C01810=1065.952,131.277,423.591,172.677,28.451,155.205
C01811=1065.946,131.028,423.611,172.676,28.448,155.204
C01812=1065.940,130.779,423.631,172.674,28.445,155.204
C01813=1065.934,130.529,423.652,172.673,28.443,155.203
C01814=1065.928,130.280,423.672,172.671,28.440,155.203
C01815=1065.922,130.032,423.692,172.669,28.438,155.203
C01816=1065.917,129.783,423.712,172.667,28.435,155.202
C01817=1065.911,129.533,423.733,172.665,28.432,155.202
C01818=1065.905,129.284,423.753,172.664,28.429,155.201
C01819=1065.899,129.035,423.772,172.662,28.426,155.201
C01820=1065.894,128.786,423.792,172.660,28.424,155.201
C01821=1065.887,128.536,423.813,172.659,28.421,155.200
C01822=1065.881,128.287,423.833,172.657,28.418,155.200
C01823=1065.876,128.038,423.853,172.656,28.416,155.200
C01824=1065.870,127.789,423.873,172.654,28.413,155.199
C01825=1065.863,127.540,423.894,172.652,28.410,155.199
C01826=1065.857,127.291,423.914,172.651,28.408,155.198
C01827=1065.851,127.007,423.936,172.648,28.404,155.198
C01828=1065.845,126.724,423.959,172.647,28.401,155.197
C01829=1065.837,126.440,423.982,172.645,28.398,155.197
C01830=1065.831,126.157,424.005,172.643,28.395,155.197
C01831=1065.826,125.907,424.025,172.641,28.392,155.196
C01832=1065.820,125.658,424.045,172.640,28.390,155.196
C01833=1065.814,125.409,424.065,172.638,28.387,155.195
C01834=1065.807,125.160,424.085,172.636,28.384,155.195
C01835=1065.802,124.911,424.106,172.635,28.381,155.195
C01836=1065.796,124.662,424.126,172.633,28.379,155.194
C01837=1065.790,124.412,424.145,172.632,28.376,155.194
C01838=1065.784,124.164,424.165,172.630,28.373,155.193
C01839=1065.779,123.914,424.186,172.628,28.370,155.193
C01840=1065.772,123.665,424.206,172.627,28.368,155.193
C01841=1065.767,123.416,424.225,172.625,28.365,155.192
C01842=1065.761,123.167,424.245,172.624,28.363,155.192
C01843=1065.755,122.918,424.265,172.622,28.360,155.191
C01844=1065.749,122.669,424.286,172.620,28.357,155.191
C01845=1065.744,122.419,424.305,172.619,28.354,155.191
C01846=1065.738,122.171,424.325,172.617,28.352,155.190
C01847=1065.732,121.922,424.345,172.616,28.349,155.190
C01848=1065.727,121.672,424.365,172.614,28.346,155.189
C01849=1065.721,121.423,424.385,172.612,28.343,155.189
C01850=1065.714,121.174,424.405,172.610,28.340,155.189
C01851=1065.708,120.924,424.424,172.608,28.337,155.188
C01852=1065.702,120.675,424.444,172.607,28.335,155.188
C01853=1065.697,120.426,424.465,172.605,28.332,155.187
C01854=1065.692,120.177,424.484,172.604,28.329,155.187
C01855=1065.686,119.928,424.504,172.602,28.326,155.187
C01856=1065.680,119.679,424.524,172.601,28.324,155.186
C01857=1065.674,119.430,424.543,172.599,28.321,155.186
C01858=1065.669,119.181,424.564,172.597,28.318,155.185
C01859=1065.663,118.931,424.583,172.596,28.315,155.185
C01860=1065.657,118.682,424.603,172.594,28.313,155.185
C01861=1065.651,118.434,424.623,172.593,28.310,155.184
C01862=1065.645,118.184,424.642,172.591,28.307,155.184
C01863=1065.639,117.935,424.662,172.589,28.304,155.183
C01864=1065.634,117.686,424.682,172.588,28.302,155.183
C01865=1065.628,117.437,424.702,172.586,28.299,155.183
C01866=1065.623,117.187,424.721,172.585,28.296,155.182
C01867=1065.617,116.939,424.741,172.583,28.293,155.182
C01868=1065.611,116.689,424.760,172.582,28.291,155.181
C01869=1065.605,116.440,424.780,172.580,28.288,155.181
C01870=1065.600,116.191,424.800,172.578,28.285,155.181
C01871=1065.594,115.942,424.820,172.577,28.282,155.180
C01872=1065.588,115.692,424.839,172.575,28.280,155.180
C01873=1065.582,115.444,424.859,172.574,28.277,155.179
C01874=1065.577,115.194,424.878,172.572,28.274,155.179
C01875=1065.571,114.945,424.898,172.571,28.271,155.178
C01876=1065.565,114.696,424.918,172.569,28.268,155.178
C01877=1065.560,114.447,424.938,172.568,28.265,155.178
C01878=1065.554,114.197,424.957,172.566,28.262,155.177
C01879=1065.548,113.948,424.977,172.564,28.260,155.177
C01880=1065.542,113.699,424.997,172.563,28.257,155.176
C01881=1065.537,113.450,425.016,172.561,28.255,155.176
C01882=1065.530,113.201,425.035,172.560,28.252,155.176
C01883=1065.524,112.952,425.054,172.558,28.249,155.175
C01884=1065.519,112.702,425.074,172.556,28.246,155.175
C01885=1065.513,112.453,425.094,172.555,28.244,155.174
C01886=1065.507,112.204,425.113,172.553,28.241,155.174
C01887=1065.501,111.955,425.132,172.552,28.238,155.174
C01888=1065.495,111.706,425.152,172.550,28.235,155.173
C01889=1065.489,111.456,425.171,172.549,28.232,155.173
C01890=1065.484,111.207,425.191,172.547,28.230,155.172
C01891=1065.477,110.923,425.213,172.545,28.227,155.172
C01892=1065.470,110.640,425.235,172.543,28.223,155.172
C01893=1065.463,110.356,425.257,172.541,28.221,155.171
C01894=1065.457,110.072,425.279,172.540,28.217,155.171
C01895=1065.450,109.823,425.298,172.538,28.215,155.170
C01896=1065.445,109.574,425.317,172.537,28.212,155.170
C01897=1065.439,109.325,425.336,172.535,28.210,155.170
C01898=1065.433,109.075,425.356,172.534,28.207,155.169
C01899=1065.427,108.826,425.376,172.532,28.204,155.169
C01900=1065.421,108.577,425.394,172.530,28.201,155.168
C01901=1065.415,108.328,425.414,172.529,28.198,155.168
C01902=1065.410,108.078,425.433,172.527,28.196,155.168
C01903=1065.404,107.830,425.452,172.526,28.193,155.167
C01904=1065.398,107.581,425.471,172.524,28.190,155.167
C01905=1065.392,107.332,425.490,172.523,28.187,155.166
C01906=1065.386,107.082,425.510,172.521,28.185,155.166
C01907=1065.381,106.833,425.529,172.519,28.182,155.166
C01908=1065.374,106.584,425.547,172.518,28.180,155.165
C01909=1065.369,106.334,425.567,172.516,28.177,155.165
C01910=1065.363,106.085,425.586,172.515,28.174,155.164
C01911=1065.357,105.836,425.606,172.513,28.171,155.164
C01912=1065.350,105.587,425.625,172.512,28.169,155.164
C01913=1065.345,105.338,425.643,172.510,28.166,155.163
C01914=1065.340,105.089,425.663,172.508,28.163,155.163
C01915=1065.334,104.839,425.682,172.507,28.160,155.162
C01916=1065.328,104.590,425.701,172.505,28.157,155.162
C01917=1065.322,104.341,425.720,172.504,28.155,155.162
C01918=1065.316,104.091,425.739,172.502,28.152,155.161
C01919=1065.310,103.842,425.758,172.501,28.149,155.161
C01920=1065.305,103.593,425.777,172.499,28.146,155.160
C01921=1065.299,103.344,425.796,172.498,28.144,155.160
C01922=1065.293,103.095,425.815,172.497,28.141,155.160
C01923=1065.287,102.845,425.834,172.495,28.138,155.159
C01924=1065.281,102.596,425.853,172.494,28.136,155.159
C01925=1065.275,102.347,425.872,172.492,28.133,155.158
C01926=1065.270,102.098,425.890,172.491,28.130,155.158
C01927=1065.264,101.849,425.910,172.489,28.127,155.158
C01928=1065.258,101.599,425.929,172.488,28.124,155.157
C01929=1065.253,101.350,425.948,172.486,28.122,155.157
C01930=1065.246,101.101,425.967,172.484,28.119,155.156
C01931=1065.241,100.852,425.986,172.483,28.116,155.156
C01932=1065.235,100.603,426.004,172.481,28.114,155.156
C01933=1065.229,100.353,426.024,172.480,28.111,155.155
C01934=1065.223,100.104,426.042,172.478,28.108,155.155
C01935=1065.217,99.855,426.061,172.477,28.106,155.154
C01936=1065.210,99.606,426.080,172.475,28.103,155.154
C01937=1065.205,99.356,426.099,172.473,28.100,155.154
C01938=1065.199,99.108,426.118,172.472,28.097,155.153
C01939=1065.193,98.859,426.137,172.470,28.094,155.153
C01940=1065.187,98.609,426.155,172.469,28.092,155.153
C01941=1065.181,98.359,426.174,172.467,28.089,155.152
C01942=1065.175,98.110,426.193,172.466,28.087,155.152
C01943=1065.170,97.862,426.212,172.464,28.084,155.151
C01944=1065.163,97.612,426.230,172.462,28.081,155.151
C01945=1065.158,97.363,426.249,172.461,28.078,155.151
C01946=1065.151,97.114,426.268,172.460,28.076,155.150
C01947=1065.146,96.864,426.287,172.459,28.073,155.150
C01948=1065.140,96.615,426.305,172.457,28.070,155.149
C01949=1065.134,96.366,426.324,172.456,28.067,155.149
C01950=1065.128,96.117,426.343,172.454,28.065,155.149
C01951=1065.122,95.867,426.361,172.452,28.062,155.148
C01952=1065.117,95.618,426.380,172.451,28.060,155.148
C01953=1065.110,95.369,426.398,172.449,28.057,155.147
C01954=1065.105,95.120,426.418,172.448,28.054,155.147
C01955=1065.098,94.836,426.439,172.446,28.051,155.147
C01956=1065.091,94.553,426.459,172.445,28.048,155.146
C01957=1065.085,94.268,426.481,172.442,28.044,155.146
C01958=1065.078,93.985,426.503,172.441,28.042,155.145
C01959=1065.072,93.736,426.520,172.439,28.039,155.145
C01960=1065.067,93.486,426.539,172.438,28.036,155.144
C01961=1065.060,93.237,426.558,172.436,28.033,155.144
C01962=1065.055,92.988,426.576,172.435,28.030,155.144
C01963=1065.049,92.739,426.595,172.433,28.028,155.143
C01964=1065.043,92.490,426.613,172.431,28.025,155.143
C01965=1065.037,92.240,426.632,172.431,28.022,155.142
C01966=1065.031,91.991,426.650,172.429,28.020,155.142
C01967=1065.026,91.742,426.670,172.428,28.017,155.142
C01968=1065.020,91.492,426.687,172.426,28.014,155.141
C01969=1065.014,91.244,426.706,172.425,28.011,155.141
C01970=1065.008,90.994,426.725,172.423,28.009,155.141
C01971=1065.002,90.745,426.743,172.421,28.006,155.140
C01972=1064.996,90.496,426.761,172.420,28.003,155.140
C01973=1064.991,90.246,426.780,172.418,28.001,155.139
C01974=1064.984,89.997,426.798,172.417,27.998,155.139
C01975=1064.979,89.748,426.816,172.415,27.995,155.139
C01976=1064.972,89.499,426.835,172.414,27.992,155.138
C01977=1064.966,89.250,426.853,172.412,27.990,155.138
C01978=1064.961,89.000,426.872,172.410,27.987,155.137
C01979=1064.955,88.751,426.890,172.409,27.985,155.137
C01980=1064.949,88.501,426.908,172.408,27.982,155.137
C01981=1064.942,88.252,426.927,172.407,27.979,155.136
C01982=1064.937,88.003,426.944,172.405,27.976,155.136
C01983=1064.931,87.754,426.963,172.404,27.974,155.135
C01984=1064.925,87.504,426.981,172.402,27.971,155.135
C01985=1064.919,87.256,427.000,172.401,27.969,155.135
C01986=1064.913,87.006,427.018,172.399,27.966,155.134
C01987=1064.906,86.757,427.036,172.397,27.963,155.134
C01988=1064.901,86.508,427.054,172.396,27.960,155.134
C01989=1064.896,86.258,427.072,172.394,27.957,155.133
C01990=1064.889,86.009,427.091,172.393,27.955,155.133
C01991=1064.884,85.760,427.109,172.391,27.952,155.132
C01992=1064.877,85.510,427.127,172.390,27.949,155.132
C01993=1064.871,85.261,427.145,172.388,27.947,155.132
C01994=1064.865,85.012,427.163,172.387,27.944,155.131
C01995=1064.859,84.763,427.181,172.386,27.942,155.131
C01996=1064.854,84.513,427.200,172.384,27.939,155.130
C01997=1064.848,84.264,427.218,172.383,27.936,155.130
C01998=1064.842,84.014,427.236,172.381,27.933,155.130
C01999=1064.836,83.766,427.254,172.380,27.930,155.129
C02000=1064.830,83.516,427.272,172.378,27.928,155.129
C02001=1064.824,83.267,427.290,172.377,27.925,155.128
C02002=1064.818,83.018,427.309,172.375,27.922,155.128
C02003=1064.812,82.768,427.326,172.373,27.920,155.128
C02004=1064.807,82.519,427.345,172.372,27.917,155.127
C02005=1064.801,82.270,427.363,172.370,27.914,155.127
C02006=1064.795,82.021,427.381,172.370,27.912,155.127
C02007=1064.789,81.771,427.399,172.368,27.909,155.126
C02008=1064.783,81.522,427.416,172.367,27.906,155.126
C02009=1064.777,81.273,427.435,172.365,27.903,155.125
C02010=1064.771,81.024,427.453,172.364,27.900,155.125
C02011=1064.765,80.774,427.470,172.362,27.898,155.125
C02012=1064.760,80.526,427.489,172.361,27.895,155.124
C02013=1064.754,80.276,427.507,172.359,27.892,155.124
C02014=1064.748,80.026,427.525,172.357,27.889,155.123
C02015=1064.743,79.777,427.543,172.356,27.887,155.123
C02016=1064.736,79.528,427.561,172.354,27.884,155.123
C02017=1064.731,79.279,427.579,172.354,27.882,155.122
C02018=1064.724,79.029,427.597,172.352,27.879,155.122
C02019=1064.718,78.746,427.618,172.350,27.875,155.121
C02020=1064.711,78.462,427.637,172.348,27.873,155.121
C02021=1064.704,78.178,427.658,172.347,27.869,155.120
C02022=1064.698,77.894,427.678,172.345,27.866,155.120
C02023=1064.692,77.645,427.697,172.344,27.864,155.120
C02024=1064.686,77.396,427.714,172.342,27.861,155.119
C02025=1064.680,77.146,427.732,172.341,27.858,155.119
C02026=1064.674,76.898,427.749,172.339,27.855,155.118
C02027=1064.668,76.648,427.767,172.338,27.853,155.118
C02028=1064.662,76.399,427.784,172.336,27.850,155.118
C02029=1064.656,76.149,427.802,172.335,27.848,155.117
C02030=1064.650,75.901,427.821,172.334,27.845,155.117
C02031=1064.644,75.651,427.839,172.332,27.842,155.117
C02032=1064.639,75.402,427.856,172.331,27.839,155.116
C02033=1064.633,75.152,427.874,172.329,27.836,155.116
C02034=1064.626,74.903,427.891,172.328,27.834,155.115
C02035=1064.620,74.654,427.909,172.326,27.831,155.115
C02036=1064.615,74.405,427.927,172.325,27.829,155.115
C02037=1064.609,74.155,427.945,172.323,27.826,155.114
C02038=1064.603,73.906,427.962,172.321,27.823,155.114
C02039=1064.597,73.656,427.980,172.321,27.820,155.113
C02040=1064.591,73.407,427.998,172.319,27.818,155.113
C02041=1064.585,73.158,428.015,172.318,27.815,155.113
C02042=1064.579,72.909,428.033,172.316,27.813,155.112
C02043=1064.573,72.659,428.050,172.315,27.810,155.112
C02044=1064.567,72.410,428.068,172.313,27.807,155.112
C02045=1064.561,72.160,428.086,172.312,27.804,155.111
C02046=1064.556,71.911,428.104,172.310,27.801,155.111
C02047=1064.549,71.662,428.120,172.309,27.799,155.110
C02048=1064.543,71.413,428.138,172.307,27.796,155.110
C02049=1064.538,71.164,428.156,172.305,27.794,155.110
C02050=1064.532,70.914,428.174,172.305,27.791,155.109
C02051=1064.526,70.665,428.191,172.303,27.788,155.109
C02052=1064.519,70.415,428.209,172.302,27.785,155.108
C02053=1064.514,70.166,428.226,172.300,27.783,155.108
C02054=1064.508,69.917,428.244,172.299,27.780,155.108
C02055=1064.502,69.667,428.261,172.297,27.777,155.107
C02056=1064.496,69.418,428.278,172.296,27.774,155.107
C02057=1064.490,69.168,428.296,172.294,27.772,155.107
C02058=1064.485,68.919,428.314,172.292,27.769,155.106
C02059=1064.478,68.670,428.331,172.292,27.767,155.106
C02060=1064.472,68.421,428.349,172.290,27.764,155.105
C02061=1064.467,68.172,428.366,172.289,27.761,155.105
C02062=1064.460,67.922,428.383,172.287,27.758,155.105
C02063=1064.455,67.673,428.400,172.286,27.756,155.104
C02064=1064.449,67.423,428.418,172.284,27.753,155.104
C02065=1064.442,67.174,428.435,172.283,27.750,155.104
C02066=1064.437,66.925,428.453,172.281,27.748,155.103
C02067=1064.431,66.676,428.471,172.280,27.745,155.103
C02068=1064.425,66.426,428.487,172.278,27.742,155.102
C02069=1064.419,66.176,428.505,172.277,27.740,155.102
C02070=1064.413,65.927,428.522,172.276,27.737,155.102
C02071=1064.407,65.679,428.539,172.274,27.734,155.101
C02072=1064.401,65.428,428.557,172.273,27.732,155.101
C02073=1064.395,65.180,428.574,172.271,27.729,155.100
C02074=1064.389,64.931,428.591,172.270,27.726,155.100
C02075=1064.383,64.681,428.609,172.268,27.723,155.100
C02076=1064.377,64.431,428.625,172.267,27.721,155.099
C02077=1064.371,64.182,428.643,172.265,27.718,155.099
C02078=1064.365,63.933,428.660,172.265,27.716,155.099
C02079=1064.360,63.683,428.677,172.263,27.713,155.098
C02080=1064.353,63.434,428.694,172.261,27.711,155.098
C02081=1064.346,63.185,428.711,172.260,27.708,155.097
C02082=1064.340,62.935,428.729,172.258,27.705,155.097
C02083=1064.334,62.651,428.748,172.257,27.702,155.097
C02084=1064.327,62.368,428.767,172.255,27.699,155.096
C02085=1064.320,62.084,428.787,172.253,27.696,155.096
C02086=1064.313,61.800,428.806,172.251,27.693,155.095
C02087=1064.306,61.551,428.823,172.250,27.691,155.095
C02088=1064.301,61.302,428.841,172.248,27.688,155.095
C02089=1064.294,61.052,428.858,172.248,27.685,155.094
C02090=1064.289,60.803,428.875,172.246,27.682,155.094
C02091=1064.282,60.553,428.892,172.245,27.680,155.094
C02092=1064.276,60.304,428.909,172.243,27.677,155.093
C02093=1064.271,60.055,428.926,172.242,27.675,155.093
C02094=1064.264,59.805,428.943,172.240,27.672,155.092
C02095=1064.258,59.556,428.960,172.238,27.670,155.092
C02096=1064.253,59.307,428.977,172.237,27.667,155.092
C02097=1064.246,59.057,428.994,172.235,27.664,155.091
C02098=1064.240,58.808,429.010,172.235,27.661,155.091
C02099=1064.234,58.559,429.028,172.233,27.659,155.091
C02100=1064.228,58.310,429.044,172.232,27.656,155.090
C02101=1064.222,58.060,429.062,172.230,27.653,155.090
C02102=1064.216,57.810,429.078,172.229,27.651,155.089
C02103=1064.210,57.562,429.095,172.227,27.648,155.089
C02104=1064.204,57.311,429.113,172.225,27.646,155.089
C02105=1064.198,57.063,429.129,172.224,27.643,155.088
C02106=1064.192,56.813,429.146,172.222,27.640,155.088
C02107=1064.186,56.564,429.163,172.222,27.637,155.088
C02108=1064.180,56.314,429.180,172.220,27.635,155.087
C02109=1064.174,56.065,429.197,172.219,27.632,155.087
C02110=1064.168,55.816,429.214,172.217,27.630,155.087
C02111=1064.162,55.566,429.231,172.216,27.627,155.086
C02112=1064.156,55.317,429.247,172.214,27.624,155.086
C02113=1064.150,55.068,429.264,172.213,27.622,155.085
C02114=1064.144,54.819,429.281,172.211,27.619,155.085
C02115=1064.138,54.569,429.297,172.210,27.616,155.085
C02116=1064.131,54.320,429.315,172.209,27.613,155.084
C02117=1064.126,54.070,429.332,172.207,27.611,155.084
C02118=1064.120,53.821,429.348,172.206,27.608,155.084
C02119=1064.114,53.572,429.365,172.204,27.606,155.083
C02120=1064.108,53.322,429.382,172.203,27.603,155.083
C02121=1064.102,53.072,429.398,172.201,27.601,155.082
C02122=1064.096,52.824,429.415,172.200,27.598,155.082
C02123=1064.091,52.574,429.432,172.198,27.595,155.082
C02124=1064.085,52.325,429.448,172.197,27.592,155.081
C02125=1064.078,52.075,429.466,172.196,27.590,155.081
C02126=1064.072,51.826,429.482,172.195,27.587,155.081
C02127=1064.067,51.576,429.499,172.193,27.584,155.080
C02128=1064.060,51.327,429.516,172.192,27.582,155.080
C02129=1064.054,51.078,429.532,172.190,27.579,155.079
C02130=1064.049,50.828,429.549,172.188,27.576,155.079
C02131=1064.042,50.579,429.566,172.187,27.574,155.079
C02132=1064.036,50.330,429.583,172.185,27.571,155.078
C02133=1064.030,50.080,429.599,172.185,27.568,155.078
C02134=1064.025,49.831,429.616,172.183,27.566,155.078
C02135=1064.019,49.582,429.633,172.182,27.563,155.077
C02136=1064.013,49.333,429.649,172.180,27.560,155.077
C02137=1064.007,49.083,429.665,172.179,27.558,155.076
C02138=1064.001,48.833,429.682,172.177,27.555,155.076
C02139=1063.995,48.584,429.699,172.176,27.552,155.076
C02140=1063.989,48.335,429.716,172.174,27.549,155.075
C02141=1063.983,48.085,429.732,172.173,27.546,155.075
C02142=1063.978,47.836,429.749,172.172,27.544,155.075
C02143=1063.972,47.586,429.765,172.170,27.542,155.074
C02144=1063.966,47.337,429.781,172.169,27.539,155.074
C02145=1063.960,47.088,429.798,172.167,27.536,155.073
C02146=1063.955,46.839,429.815,172.166,27.533,155.073
C02147=1063.948,46.555,429.834,172.164,27.530,155.073
C02148=1063.940,46.270,429.852,172.163,27.527,155.072
C02149=1063.933,45.986,429.871,172.162,27.524,155.072
C02150=1063.927,45.702,429.890,172.160,27.521,155.071
C02151=1063.922,45.453,429.907,172.159,27.518,155.071
C02152=1063.916,45.203,429.923,172.157,27.516,155.070
C02153=1063.910,44.954,429.939,172.156,27.513,155.070
C02154=1063.904,44.704,429.956,172.154,27.510,155.070
C02155=1063.898,44.455,429.972,172.152,27.508,155.069
C02156=1063.893,44.205,429.989,172.151,27.505,155.069
C02157=1063.886,43.957,430.006,172.149,27.502,155.069
C02158=1063.880,43.707,430.022,172.148,27.499,155.068
C02159=1063.874,43.458,430.038,172.147,27.497,155.068
C02160=1063.869,43.209,430.054,172.146,27.494,155.068
C02161=1063.863,42.959,430.071,172.144,27.492,155.067
C02162=1063.856,42.709,430.087,172.143,27.489,155.067
C02163=1063.850,42.460,430.104,172.141,27.486,155.066
C02164=1063.844,42.211,430.120,172.140,27.484,155.066
C02165=1063.838,41.961,430.136,172.138,27.481,155.066
C02166=1063.832,41.712,430.152,172.137,27.478,155.065
C02167=1063.826,41.463,430.169,172.136,27.476,155.065
C02168=1063.820,41.213,430.185,172.134,27.473,155.065
C02169=1063.814,40.964,430.201,172.133,27.470,155.064
C02170=1063.808,40.715,430.217,172.131,27.468,155.064
C02171=1063.802,40.465,430.234,172.130,27.465,155.064
C02172=1063.797,40.215,430.249,172.128,27.462,155.063
C02173=1063.791,39.966,430.265,172.127,27.460,155.063
C02174=1063.785,39.717,430.282,172.125,27.457,155.062
C02175=1063.779,39.467,430.298,172.124,27.455,155.062
C02176=1063.773,39.218,430.314,172.123,27.452,155.062
C02177=1063.767,38.968,430.330,172.122,27.449,155.061
C02178=1063.761,38.719,430.347,172.120,27.447,155.061
C02179=1063.755,38.470,430.363,172.119,27.444,155.061
C02180=1063.749,38.220,430.379,172.117,27.441,155.060
C02181=1063.743,37.971,430.395,172.116,27.438,155.060
C02182=1063.738,37.721,430.411,172.114,27.436,155.060
C02183=1063.731,37.472,430.427,172.113,27.433,155.059
C02184=1063.725,37.223,430.443,172.111,27.431,155.059
C02185=1063.719,36.973,430.459,172.110,27.429,155.058
C02186=1063.713,36.724,430.475,172.109,27.426,155.058
C02187=1063.707,36.475,430.492,172.107,27.423,155.058
C02188=1063.701,36.225,430.507,172.106,27.421,155.057
C02189=1063.695,35.976,430.523,172.104,27.418,155.057
C02190=1063.689,35.726,430.539,172.103,27.416,155.057
C02191=1063.683,35.477,430.555,172.101,27.413,155.056
C02192=1063.677,35.228,430.572,172.100,27.410,155.056
C02193=1063.671,34.978,430.587,172.098,27.408,155.056
C02194=1063.665,34.729,430.603,172.098,27.405,155.055
C02195=1063.659,34.479,430.619,172.096,27.402,155.055
C02196=1063.653,34.230,430.635,172.094,27.400,155.055
C02197=1063.646,33.980,430.650,172.093,27.397,155.054
C02198=1063.640,33.731,430.667,172.091,27.394,155.054
C02199=1063.634,33.482,430.683,172.090,27.392,155.053
C02200=1063.629,33.232,430.698,172.088,27.389,155.053
C02201=1063.622,32.983,430.714,172.087,27.386,155.053
C02202=1063.616,32.733,430.730,172.086,27.384,155.052
C02203=1063.610,32.484,430.747,172.085,27.382,155.052
C02204=1063.605,32.234,430.762,172.083,27.379,155.052
C02205=1063.598,31.985,430.778,172.082,27.376,155.051
C02206=1063.592,31.736,430.794,172.080,27.374,155.051
C02207=1063.586,31.486,430.810,172.079,27.371,155.051
C02208=1063.580,31.236,430.826,172.077,27.368,155.050
C02209=1063.574,30.987,430.842,172.076,27.366,155.050
C02210=1063.569,30.738,430.857,172.074,27.363,155.050
C02211=1063.561,30.454,430.875,172.073,27.360,155.049
C02212=1063.555,30.170,430.893,172.071,27.357,155.049
C02213=1063.548,29.885,430.911,172.070,27.354,155.048
C02214=1063.541,29.601,430.929,172.068,27.351,155.048
C02215=1063.535,29.352,430.945,172.067,27.349,155.048
C02216=1063.529,29.102,430.960,172.065,27.346,155.047
C02217=1063.523,28.853,430.977,172.064,27.344,155.047
C02218=1063.517,28.603,430.992,172.062,27.341,155.046
C02219=1063.511,28.354,431.008,172.061,27.338,155.046
C02220=1063.506,28.105,431.023,172.059,27.336,155.046
C02221=1063.499,27.855,431.039,172.058,27.334,155.046
C02222=1063.493,27.605,431.054,172.057,27.331,155.045
C02223=1063.487,27.356,431.070,172.055,27.328,155.045
C02224=1063.481,27.106,431.086,172.054,27.326,155.044
C02225=1063.474,26.857,431.101,172.052,27.323,155.044
C02226=1063.469,26.607,431.117,172.051,27.321,155.044
C02227=1063.463,26.358,431.133,172.049,27.318,155.043
C02228=1063.456,26.108,431.148,172.048,27.315,155.043
C02229=1063.451,25.860,431.164,172.046,27.313,155.043
C02230=1063.445,25.610,431.179,172.046,27.310,155.042
C02231=1063.439,25.361,431.195,172.044,27.308,155.042
C02232=1063.432,25.111,431.210,172.043,27.305,155.042
C02233=1063.426,24.862,431.226,172.041,27.303,155.041
C02234=1063.420,24.612,431.241,172.039,27.300,155.041
C02235=1063.414,24.363,431.257,172.038,27.298,155.041
C02236=1063.408,24.114,431.272,172.036,27.295,155.040
C02237=1063.403,23.864,431.288,172.035,27.292,155.040
C02238=1063.396,23.615,431.303,172.033,27.290,155.040
C02239=1063.390,23.365,431.319,172.032,27.287,155.039
C02240=1063.384,23.116,431.334,172.031,27.285,155.039
C02241=1063.378,22.866,431.350,172.030,27.282,155.039
C02242=1063.372,22.617,431.365,172.028,27.280,155.038
C02243=1063.366,22.368,431.381,172.027,27.277,155.038
C02244=1063.360,22.118,431.396,172.025,27.274,155.037
C02245=1063.354,21.868,431.411,172.024,27.272,155.037
C02246=1063.347,21.619,431.427,172.022,27.269,155.037
C02247=1063.342,21.370,431.442,172.021,27.267,155.037
C02248=1063.336,21.120,431.457,172.019,27.264,155.036
C02249=1063.330,20.871,431.473,172.018,27.262,155.036
C02250=1063.324,20.621,431.488,172.017,27.259,155.035
C02251=1063.318,20.371,431.504,172.015,27.257,155.035
C02252=1063.312,20.123,431.519,172.014,27.254,155.035
C02253=1063.306,19.873,431.534,172.012,27.252,155.035
C02254=1063.300,19.623,431.550,172.011,27.249,155.034
C02255=1063.293,19.374,431.565,172.009,27.246,155.034
C02256=1063.287,19.124,431.580,172.008,27.244,155.033
C02257=1063.282,18.875,431.595,172.006,27.241,155.033
C02258=1063.275,18.625,431.610,172.005,27.238,155.033
C02259=1063.270,18.376,431.627,172.004,27.236,155.033
C02260=1063.263,18.126,431.642,172.003,27.234,155.032
C02261=1063.257,17.877,431.656,172.001,27.231,155.032
C02262=1063.252,17.628,431.672,171.999,27.229,155.031
C02263=1063.245,17.378,431.687,171.998,27.226,155.031
C02264=1063.239,17.129,431.702,171.996,27.223,155.031
C02265=1063.234,16.880,431.717,171.995,27.221,155.031
C02266=1063.227,16.630,431.732,171.993,27.218,155.030
C02267=1063.221,16.380,431.747,171.992,27.216,155.030
C02268=1063.215,16.130,431.763,171.990,27.213,155.029
C02269=1063.209,15.881,431.777,171.990,27.211,155.029
C02270=1063.203,15.632,431.793,171.988,27.208,155.029
C02271=1063.197,15.382,431.809,171.987,27.206,155.028
C02272=1063.191,15.133,431.824,171.985,27.203,155.028
C02273=1063.185,14.884,431.838,171.984,27.201,155.028
C02274=1063.179,14.634,431.854,171.982,27.198,155.027
C02275=1063.172,14.351,431.871,171.981,27.195,155.027
C02276=1063.165,14.069,431.887,171.979,27.192,155.027
C02277=1063.158,13.786,431.905,171.978,27.190,155.026
C02278=1063.151,13.503,431.922,171.975,27.187,155.026
C02279=1063.145,13.254,431.937,171.974,27.184,155.026
C02280=1063.139,13.004,431.952,171.973,27.182,155.025
C02281=1063.132,12.754,431.967,171.972,27.179,155.025
C02282=1063.126,12.505,431.982,171.970,27.177,155.025
C02283=1063.120,12.256,431.996,171.968,27.175,155.024
C02284=1063.114,12.006,432.011,171.967,27.172,155.024
C02285=1063.108,11.757,432.026,171.965,27.170,155.024
C02286=1063.103,11.507,432.041,171.964,27.167,155.023
C02287=1063.096,11.258,432.056,171.962,27.165,155.023
C02288=1063.090,11.008,432.071,171.961,27.162,155.023
C02289=1063.083,10.758,432.086,171.959,27.159,155.022
C02290=1063.078,10.509,432.101,171.958,27.157,155.022
C02291=1063.071,10.260,432.116,171.956,27.155,155.022
C02292=1063.065,10.010,432.131,171.956,27.152,155.021
C02293=1063.059,9.761,432.145,171.954,27.150,155.021
C02294=1063.053,9.511,432.160,171.952,27.148,155.021
C02295=1063.046,9.262,432.175,171.951,27.145,155.021
C02296=1063.040,9.013,432.190,171.949,27.143,155.020
C02297=1063.035,8.763,432.205,171.948,27.140,155.020
C02298=1063.028,8.513,432.220,171.946,27.137,155.020
C02299=1063.023,8.264,432.234,171.945,27.135,155.019
C02300=1063.017,8.014,432.249,171.943,27.132,155.019
C02301=1063.010,7.764,432.264,171.942,27.130,155.019
C02302=1063.004,7.515,432.278,171.940,27.128,155.018
C02303=1062.998,7.266,432.293,171.940,27.125,155.018
C02304=1062.992,7.017,432.308,171.938,27.123,155.018
C02305=1062.986,6.767,432.323,171.936,27.121,155.017
C02306=1062.980,6.517,432.338,171.935,27.118,155.017
C02307=1062.974,6.268,432.352,171.933,27.115,155.017
C02308=1062.968,6.018,432.367,171.932,27.113,155.017
C02309=1062.961,5.769,432.382,171.930,27.110,155.016
C02310=1062.955,5.520,432.396,171.929,27.108,155.016
C02311=1062.949,5.270,432.411,171.927,27.105,155.015
C02312=1062.943,5.021,432.426,171.926,27.103,155.015
C02313=1062.937,4.771,432.440,171.924,27.101,155.015
C02314=1062.931,4.522,432.455,171.923,27.098,155.015
C02315=1062.925,4.272,432.469,171.921,27.096,155.014
C02316=1062.919,4.022,432.485,171.920,27.094,155.014
C02317=1062.914,3.773,432.500,171.919,27.091,155.014
C02318=1062.908,3.523,432.514,171.917,27.088,155.013
C02319=1062.902,3.274,432.528,171.916,27.086,155.013
C02320=1062.895,3.024,432.543,171.914,27.083,155.013
C02321=1062.890,2.775,432.558,171.913,27.081,155.012
C02322=1062.884,2.525,432.572,171.911,27.079,155.012
C02323=1062.877,2.275,432.587,171.910,27.076,155.012
C02324=1062.871,2.026,432.602,171.908,27.074,155.011
C02325=1062.865,1.777,432.617,171.907,27.071,155.011
C02326=1062.860,1.527,432.630,171.905,27.068,155.011
C02327=1062.853,1.278,432.645,171.904,27.066,155.011
C02328=1062.847,1.029,432.660,171.903,27.064,155.010
C02329=1062.841,0.778,432.674,171.902,27.061,155.010
C02330=1062.835,0.529,432.689,171.900,27.059,155.010
C02331=1062.829,0.280,432.704,171.899,27.056,155.009
C02332=1062.824,0.030,432.718,171.897,27.054,155.009
C02333=1062.817,-0.220,432.733,171.895,27.052,155.009
C02334=1062.811,-0.469,432.747,171.894,27.049,155.008
C02335=1062.805,-0.719,432.761,171.892,27.046,155.008
C02336=1062.800,-0.968,432.776,171.891,27.044,155.008
C02337=1062.793,-1.217,432.791,171.889,27.041,155.007
C02338=1062.787,-1.467,432.804,171.888,27.039,155.007
C02339=1062.781,-1.747,432.821,171.886,27.036,155.007
C02340=1062.774,-2.029,432.837,171.885,27.034,155.006
C02341=1062.767,-2.309,432.854,171.883,27.031,155.006
C02342=1062.761,-2.590,432.869,171.882,27.028,155.006
C02343=1062.754,-2.839,432.884,171.880,27.026,155.005
C02344=1062.749,-3.089,432.898,171.879,27.023,155.005
C02345=1062.743,-3.339,432.913,171.877,27.021,155.005
C02346=1062.737,-3.588,432.927,171.876,27.018,155.004
C02347=1062.730,-3.838,432.941,171.874,27.016,155.004
C02348=1062.724,-4.087,432.955,171.872,27.014,155.004
C02349=1062.718,-4.337,432.970,171.871,27.011,155.003
C02350=1062.712,-4.586,432.983,171.869,27.009,155.003
C02351=1062.705,-4.836,432.998,171.868,27.006,155.003
C02352=1062.700,-5.085,433.012,171.866,27.004,155.003
C02353=1062.693,-5.335,433.027,171.865,27.002,155.002
C02354=1062.687,-5.584,433.040,171.863,27.000,155.002
C02355=1062.681,-5.834,433.055,171.862,26.997,155.002
C02356=1062.676,-6.083,433.069,171.860,26.994,155.001
C02357=1062.668,-6.333,433.084,171.860,26.992,155.001
C02358=1062.663,-6.582,433.098,171.858,26.990,155.001
C02359=1062.657,-6.833,433.112,171.856,26.988,155.001
C02360=1062.650,-7.081,433.126,171.855,26.986,155.000
C02361=1062.645,-7.331,433.140,171.853,26.983,155.000
C02362=1062.638,-7.581,433.155,171.852,26.980,155.000
C02363=1062.632,-7.830,433.168,171.850,26.978,154.999
C02364=1062.626,-8.079,433.183,171.849,26.976,154.999
C02365=1062.620,-8.329,433.197,171.847,26.974,154.999
C02366=1062.614,-8.579,433.210,171.846,26.971,154.999
C02367=1062.608,-8.828,433.225,171.844,26.969,154.998
C02368=1062.602,-9.078,433.239,171.842,26.967,154.998
C02369=1062.596,-9.327,433.252,171.841,26.964,154.998
C02370=1062.590,-9.576,433.267,171.839,26.962,154.997
C02371=1062.584,-9.827,433.281,171.838,26.959,154.997
C02372=1062.577,-10.076,433.294,171.836,26.957,154.997
C02373=1062.572,-10.325,433.309,171.835,26.955,154.997
C02374=1062.565,-10.575,433.323,171.833,26.952,154.996
C02375=1062.559,-10.824,433.336,171.832,26.950,154.996
C02376=1062.553,-11.074,433.351,171.831,26.947,154.996
C02377=1062.547,-11.323,433.365,171.830,26.945,154.995
C02378=1062.541,-11.573,433.379,171.828,26.943,154.995
C02379=1062.535,-11.823,433.394,171.826,26.941,154.995
C02380=1062.529,-12.072,433.407,171.825,26.938,154.995
C02381=1062.523,-12.321,433.421,171.823,26.936,154.994
C02382=1062.517,-12.572,433.435,171.822,26.934,154.994
C02383=1062.511,-12.820,433.449,171.820,26.931,154.994
C02384=1062.505,-13.070,433.463,171.819,26.929,154.993
C02385=1062.498,-13.320,433.476,171.817,26.926,154.993
C02386=1062.493,-13.570,433.490,171.816,26.924,154.993
C02387=1062.487,-13.819,433.504,171.814,26.922,154.993
C02388=1062.480,-14.068,433.518,171.813,26.919,154.992
C02389=1062.475,-14.318,433.532,171.811,26.917,154.992
C02390=1062.469,-14.567,433.546,171.809,26.915,154.992
C02391=1062.463,-14.818,433.560,171.808,26.913,154.992
C02392=1062.457,-15.067,433.574,171.806,26.910,154.991
C02393=1062.451,-15.316,433.588,171.805,26.908,154.991
C02394=1062.444,-15.566,433.601,171.803,26.906,154.991
C02395=1062.438,-15.815,433.615,171.802,26.903,154.990
C02396=1062.432,-16.065,433.628,171.800,26.901,154.990
C02397=1062.426,-16.315,433.643,171.799,26.899,154.990
C02398=1062.420,-16.564,433.656,171.798,26.897,154.990
C02399=1062.414,-16.814,433.670,171.796,26.894,154.989
C02400=1062.407,-17.064,433.683,171.795,26.892,154.989
C02401=1062.401,-17.312,433.697,171.793,26.890,154.989
C02402=1062.395,-17.562,433.711,171.792,26.888,154.989
C02403=1062.386,-17.913,433.730,171.789,26.884,154.988
C02404=1062.378,-18.262,433.749,171.787,26.881,154.988
C02405=1062.369,-18.612,433.768,171.785,26.878,154.987
C02406=1062.361,-18.962,433.788,171.783,26.875,154.987
C02407=1062.355,-19.211,433.801,171.782,26.872,154.987
C02408=1062.349,-19.461,433.815,171.780,26.870,154.987
C02409=1062.342,-19.710,433.829,171.778,26.868,154.986
C02410=1062.336,-19.960,433.842,171.777,26.866,154.986
C02411=1062.330,-20.210,433.856,171.775,26.864,154.986
C02412=1062.324,-20.459,433.869,171.774,26.862,154.986
C02413=1062.318,-20.709,433.883,171.772,26.859,154.985
C02414=1062.312,-20.958,433.896,171.771,26.857,154.985
C02415=1062.305,-21.208,433.910,171.769,26.855,154.985
C02416=1062.299,-21.457,433.923,171.767,26.852,154.985
C02417=1062.294,-21.707,433.937,171.766,26.850,154.984
C02418=1062.288,-21.956,433.950,171.764,26.848,154.984
C02419=1062.281,-22.206,433.965,171.763,26.845,154.984
C02420=1062.275,-22.456,433.978,171.761,26.843,154.983
C02421=1062.269,-22.705,433.991,171.760,26.841,154.983
C02422=1062.264,-22.955,434.004,171.758,26.839,154.983
C02423=1062.258,-23.204,434.018,171.757,26.836,154.983
C02424=1062.251,-23.454,434.031,171.755,26.834,154.982
C02425=1062.245,-23.704,434.045,171.753,26.832,154.982
C02426=1062.239,-23.953,434.058,171.752,26.830,154.982
C02427=1062.233,-24.202,434.072,171.750,26.828,154.982
C02428=1062.227,-24.452,434.086,171.749,26.825,154.981
C02429=1062.221,-24.701,434.099,171.747,26.823,154.981
C02430=1062.214,-24.951,434.112,171.746,26.821,154.981
C02431=1062.210,-25.165,434.124,171.745,26.819,154.981
C02432=1062.204,-25.380,434.135,171.743,26.817,154.980
C02433=1062.199,-25.594,434.147,171.742,26.815,154.980
C02434=1062.194,-25.809,434.158,171.741,26.813,154.980
C02435=1062.188,-26.022,434.170,171.739,26.812,154.980
C02436=1062.184,-26.236,434.181,171.738,26.809,154.980
C02437=1062.179,-26.451,434.192,171.736,26.808,154.979
C02438=1062.173,-26.665,434.204,171.736,26.806,154.979
C02439=1062.168,-26.914,434.218,171.734,26.803,154.979
C02440=1062.162,-27.164,434.231,171.732,26.801,154.979
C02441=1062.156,-27.414,434.244,171.731,26.799,154.978
C02442=1062.149,-27.664,434.257,171.729,26.797,154.978
C02443=1062.142,-27.913,434.271,171.728,26.795,154.978
C02444=1062.137,-28.163,434.283,171.726,26.792,154.978
C02445=1062.130,-28.412,434.297,171.725,26.791,154.977
C02446=1062.124,-28.661,434.310,171.723,26.788,154.977
C02447=1062.117,-28.911,434.323,171.721,26.786,154.977
C02448=1062.112,-29.161,434.337,171.720,26.784,154.977
C02449=1062.106,-29.411,434.350,171.718,26.782,154.977
C02450=1062.100,-29.660,434.363,171.717,26.780,154.976
C02451=1062.094,-29.909,434.376,171.715,26.777,154.976
C02452=1062.088,-30.159,434.389,171.713,26.776,154.976
C02453=1062.081,-30.408,434.402,171.712,26.773,154.976
C02454=1062.075,-30.658,434.416,171.710,26.771,154.975
C02455=1062.069,-30.908,434.428,171.709,26.769,154.975
C02456=1062.062,-31.157,434.442,171.707,26.767,154.975
C02457=1062.056,-31.407,434.455,171.706,26.765,154.975
C02458=1062.050,-31.657,434.467,171.704,26.762,154.974
C02459=1062.044,-31.906,434.481,171.702,26.761,154.974
C02460=1062.038,-32.156,434.493,171.701,26.758,154.974
C02461=1062.033,-32.405,434.507,171.699,26.756,154.974
C02462=1062.027,-32.655,434.520,171.698,26.754,154.973
C02463=1062.020,-32.905,434.533,171.696,26.752,154.973
C02464=1062.014,-33.154,434.547,171.695,26.750,154.973
C02465=1062.008,-33.404,434.560,171.693,26.747,154.973
C02466=1062.002,-33.654,434.572,171.691,26.746,154.973
C02467=1061.995,-33.931,434.587,171.690,26.743,154.972
C02468=1061.988,-34.210,434.602,171.688,26.741,154.972
C02469=1061.981,-34.488,434.615,171.686,26.739,154.972
C02470=1061.975,-34.767,434.630,171.684,26.736,154.972
C02471=1061.968,-35.016,434.644,171.683,26.734,154.971
C02472=1061.962,-35.266,434.656,171.681,26.732,154.971
C02473=1061.956,-35.516,434.669,171.679,26.730,154.971
C02474=1061.950,-35.765,434.682,171.678,26.728,154.971
C02475=1061.944,-36.015,434.695,171.676,26.725,154.970
C02476=1061.938,-36.265,434.708,171.675,26.724,154.970
C02477=1061.932,-36.514,434.721,171.673,26.721,154.970
C02478=1061.926,-36.764,434.734,171.672,26.719,154.970
C02479=1061.920,-37.013,434.747,171.670,26.717,154.970
C02480=1061.914,-37.263,434.759,171.668,26.715,154.969
C02481=1061.908,-37.512,434.773,171.667,26.713,154.969
C02482=1061.902,-37.762,434.785,171.665,26.711,154.969
C02483=1061.896,-38.011,434.799,171.664,26.709,154.969
C02484=1061.890,-38.261,434.811,171.662,26.706,154.968
C02485=1061.884,-38.511,434.824,171.660,26.705,154.968
C02486=1061.878,-38.760,434.837,171.659,26.702,154.968
C02487=1061.872,-39.010,434.849,171.657,26.701,154.968
C02488=1061.865,-39.259,434.863,171.656,26.698,154.968
C02489=1061.859,-39.509,434.875,171.654,26.697,154.967
C02490=1061.853,-39.759,434.887,171.653,26.694,154.967
C02491=1061.847,-40.008,434.901,171.651,26.692,154.967
C02492=1061.841,-40.258,434.913,171.649,26.690,154.967
C02493=1061.835,-40.507,434.926,171.648,26.688,154.967
C02494=1061.828,-40.757,434.938,171.646,26.686,154.966
C02495=1061.822,-41.007,434.951,171.645,26.684,154.966
C02496=1061.816,-41.256,434.964,171.643,26.682,154.966
C02497=1061.810,-41.506,434.977,171.641,26.680,154.966
C02498=1061.804,-41.756,434.989,171.640,26.678,154.966
C02499=1061.797,-42.005,435.002,171.638,26.676,154.965
C02500=1061.791,-42.255,435.014,171.637,26.674,154.965
C02501=1061.785,-42.505,435.027,171.635,26.672,154.965
C02502=1061.779,-42.754,435.040,171.633,26.670,154.965
C02503=1061.772,-43.003,435.052,171.632,26.668,154.965
C02504=1061.766,-43.253,435.065,171.630,26.666,154.964
C02505=1061.761,-43.503,435.077,171.629,26.664,154.964
C02506=1061.754,-43.752,435.091,171.627,26.662,154.964
C02507=1061.748,-44.002,435.103,171.625,26.660,154.964
C02508=1061.742,-44.252,435.115,171.624,26.658,154.963
C02509=1061.736,-44.502,435.128,171.622,26.656,154.963
C02510=1061.730,-44.751,435.141,171.620,26.654,154.963
C02511=1061.724,-45.001,435.154,171.619,26.652,154.963
C02512=1061.717,-45.250,435.165,171.617,26.650,154.963
C02513=1061.712,-45.500,435.178,171.616,26.648,154.963
C02514=1061.706,-45.750,435.190,171.614,26.646,154.962
C02515=1061.700,-45.999,435.203,171.613,26.644,154.962
C02516=1061.693,-46.248,435.215,171.611,26.642,154.962
C02517=1061.687,-46.498,435.228,171.609,26.641,154.962
C02518=1061.681,-46.748,435.241,171.608,26.638,154.962
C02519=1061.675,-46.998,435.253,171.606,26.637,154.961
C02520=1061.668,-47.247,435.266,171.605,26.634,154.961
C02521=1061.662,-47.497,435.278,171.603,26.633,154.961
C02522=1061.657,-47.746,435.291,171.601,26.631,154.961
C02523=1061.651,-47.996,435.302,171.600,26.628,154.961
C02524=1061.645,-48.245,435.315,171.598,26.627,154.960
C02525=1061.639,-48.495,435.328,171.597,26.624,154.960
C02526=1061.633,-48.745,435.340,171.595,26.623,154.960
C02527=1061.626,-48.995,435.352,171.593,26.621,154.960
C02528=1061.621,-49.244,435.364,171.592,26.619,154.960
C02529=1061.615,-49.493,435.378,171.590,26.617,154.959
C02530=1061.608,-49.743,435.390,171.588,26.615,154.959
C02531=1061.602,-50.022,435.404,171.586,26.613,154.959
C02532=1061.595,-50.301,435.417,171.584,26.610,154.959
C02533=1061.588,-50.580,435.431,171.583,26.609,154.959
C02534=1061.580,-50.859,435.445,171.580,26.606,154.959
C02535=1061.574,-51.108,435.457,171.579,26.604,154.958
C02536=1061.569,-51.357,435.469,171.577,26.603,154.958
C02537=1061.562,-51.607,435.481,171.575,26.601,154.958
C02538=1061.556,-51.857,435.494,171.574,26.599,154.958
C02539=1061.549,-52.106,435.506,171.572,26.597,154.958
C02540=1061.543,-52.356,435.518,171.570,26.595,154.958
C02541=1061.537,-52.606,435.530,171.569,26.593,154.957
C02542=1061.530,-52.856,435.541,171.567,26.592,154.957
C02543=1061.525,-53.105,435.554,171.565,26.590,154.957
C02544=1061.518,-53.355,435.566,171.564,26.588,154.957
C02545=1061.512,-53.604,435.577,171.562,26.586,154.957
C02546=1061.506,-53.854,435.590,171.561,26.584,154.957
C02547=1061.499,-54.104,435.602,171.559,26.582,154.956
C02548=1061.493,-54.354,435.615,171.557,26.581,154.956
C02549=1061.487,-54.603,435.627,171.556,26.579,154.956
C02550=1061.481,-54.852,435.638,171.554,26.577,154.956
C02551=1061.475,-55.102,435.651,171.552,26.575,154.956
C02552=1061.468,-55.352,435.663,171.551,26.574,154.956
C02553=1061.462,-55.602,435.675,171.549,26.572,154.956
C02554=1061.456,-55.852,435.686,171.548,26.570,154.955
C02555=1061.450,-56.101,435.698,171.546,26.568,154.955
C02556=1061.444,-56.350,435.711,171.544,26.566,154.955
C02557=1061.437,-56.600,435.723,171.543,26.564,154.955
C02558=1061.431,-56.850,435.734,171.541,26.563,154.955
C02559=1061.425,-57.100,435.747,171.539,26.561,154.955
C02560=1061.419,-57.348,435.759,171.538,26.559,154.954
C02561=1061.412,-57.599,435.770,171.536,26.557,154.954
C02562=1061.406,-57.848,435.782,171.534,26.556,154.954
C02563=1061.400,-58.098,435.794,171.532,26.554,154.954
C02564=1061.394,-58.347,435.807,171.530,26.552,154.954
C02565=1061.388,-58.597,435.819,171.529,26.550,154.954
C02566=1061.381,-58.847,435.830,171.527,26.548,154.953
C02567=1061.376,-59.097,435.842,171.525,26.546,154.953
C02568=1061.370,-59.346,435.854,171.524,26.544,154.953
C02569=1061.363,-59.595,435.866,171.522,26.543,154.953
C02570=1061.357,-59.846,435.878,171.520,26.541,154.953
C02571=1061.351,-60.095,435.890,171.519,26.539,154.953
C02572=1061.345,-60.344,435.901,171.517,26.538,154.953
C02573=1061.339,-60.594,435.914,171.515,26.536,154.952
C02574=1061.332,-60.844,435.925,171.514,26.534,154.952
C02575=1061.326,-61.093,435.937,171.512,26.532,154.952
C02576=1061.320,-61.343,435.949,171.511,26.531,154.952
C02577=1061.314,-61.593,435.961,171.509,26.529,154.952
C02578=1061.307,-61.843,435.972,171.507,26.527,154.952
C02579=1061.301,-62.092,435.984,171.506,26.525,154.952
C02580=1061.295,-62.342,435.997,171.504,26.524,154.951
C02581=1061.289,-62.592,436.008,171.502,26.522,154.951
C02582=1061.283,-62.841,436.019,171.501,26.520,154.951
C02583=1061.277,-63.091,436.032,171.499,26.518,154.951
C02584=1061.271,-63.341,436.043,171.497,26.517,154.951
C02585=1061.265,-63.590,436.055,171.496,26.515,154.951
C02586=1061.259,-63.840,436.067,171.494,26.513,154.951
C02587=1061.253,-64.090,436.079,171.492,26.511,154.951
C02588=1061.246,-64.339,436.090,171.490,26.509,154.950
C02589=1061.240,-64.589,436.101,171.488,26.508,154.950
C02590=1061.235,-64.838,436.114,171.487,26.506,154.950
C02591=1061.228,-65.087,436.126,171.485,26.504,154.950
C02592=1061.222,-65.338,436.137,171.483,26.503,154.950
C02593=1061.217,-65.587,436.149,171.482,26.501,154.950
C02594=1061.210,-65.837,436.160,171.480,26.500,154.950
C02595=1061.203,-66.117,436.173,171.478,26.497,154.949
C02596=1061.196,-66.396,436.186,171.477,26.496,154.949
C02597=1061.189,-66.677,436.199,171.474,26.494,154.949
C02598=1061.183,-66.957,436.213,171.472,26.492,154.949
C02599=1061.177,-67.208,436.224,171.471,26.490,154.949
C02600=1061.171,-67.456,436.236,171.469,26.488,154.949
C02601=1061.164,-67.706,436.248,171.468,26.487,154.949
C02602=1061.159,-67.956,436.259,171.466,26.485,154.948
C02603=1061.152,-68.205,436.271,171.464,26.483,154.948
C02604=1061.147,-68.455,436.282,171.463,26.481,154.948
C02605=1061.140,-68.705,436.293,171.461,26.480,154.948
C02606=1061.134,-68.954,436.305,171.459,26.478,154.948
C02607=1061.129,-69.204,436.317,171.458,26.477,154.948
C02608=1061.122,-69.454,436.329,171.456,26.475,154.948
C02609=1061.116,-69.704,436.340,171.453,26.473,154.948
C02610=1061.110,-69.953,436.351,171.452,26.471,154.947
C02611=1061.105,-70.203,436.363,171.450,26.470,154.947
C02612=1061.098,-70.452,436.375,171.448,26.468,154.947
C02613=1061.092,-70.702,436.386,171.447,26.467,154.947
C02614=1061.086,-70.952,436.397,171.445,26.465,154.947
C02615=1061.081,-71.201,436.409,171.443,26.463,154.947
C02616=1061.074,-71.452,436.420,171.442,26.461,154.947
C02617=1061.068,-71.700,436.432,171.440,26.460,154.947
C02618=1061.062,-71.951,436.443,171.438,26.458,154.946
C02619=1061.056,-72.200,436.454,171.437,26.456,154.946
C02620=1061.050,-72.450,436.467,171.435,26.455,154.946
C02621=1061.044,-72.699,436.478,171.433,26.453,154.946
C02622=1061.038,-72.949,436.490,171.432,26.452,154.946
C02623=1061.032,-73.199,436.500,171.430,26.450,154.946
C02624=1061.026,-73.449,436.512,171.428,26.448,154.946
C02625=1061.020,-73.698,436.524,171.427,26.447,154.946
C02626=1061.014,-73.948,436.535,171.425,26.445,154.946
C02627=1061.008,-74.198,436.546,171.423,26.443,154.945
C02628=1061.002,-74.448,436.557,171.422,26.442,154.945
C02629=1060.996,-74.697,436.569,171.419,26.440,154.945
C02630=1060.990,-74.947,436.580,171.417,26.439,154.945
C02631=1060.984,-75.196,436.591,171.416,26.437,154.945
C02632=1060.977,-75.446,436.603,171.414,26.436,154.945
C02633=1060.971,-75.695,436.614,171.412,26.434,154.945
C02634=1060.964,-75.945,436.624,171.411,26.433,154.945
C02635=1060.959,-76.195,436.635,171.409,26.431,154.945
C02636=1060.952,-76.445,436.647,171.407,26.429,154.945
C02637=1060.946,-76.694,436.658,171.406,26.428,154.945
C02638=1060.941,-76.943,436.669,171.404,26.426,154.944
C02639=1060.934,-77.194,436.680,171.402,26.425,154.944
C02640=1060.928,-77.443,436.691,171.401,26.423,154.944
C02641=1060.922,-77.693,436.703,171.399,26.422,154.944
C02642=1060.916,-77.942,436.714,171.397,26.421,154.944
C02643=1060.910,-78.192,436.725,171.396,26.419,154.944
C02644=1060.904,-78.442,436.736,171.394,26.418,154.944
C02645=1060.898,-78.692,436.747,171.392,26.416,154.944
C02646=1060.892,-78.941,436.758,171.389,26.414,154.944
C02647=1060.885,-79.191,436.770,171.388,26.413,154.944
C02648=1060.880,-79.440,436.781,171.386,26.411,154.944
C02649=1060.874,-79.690,436.792,171.384,26.410,154.944
C02650=1060.867,-79.940,436.803,171.383,26.408,154.943
C02651=1060.861,-80.189,436.813,171.381,26.407,154.943
C02652=1060.855,-80.440,436.825,171.379,26.406,154.943
C02653=1060.849,-80.689,436.836,171.378,26.404,154.943
C02654=1060.842,-80.939,436.846,171.376,26.403,154.943
C02655=1060.836,-81.188,436.857,171.374,26.401,154.943
C02656=1060.830,-81.439,436.868,171.372,26.400,154.943
C02657=1060.824,-81.687,436.880,171.371,26.399,154.943
C02658=1060.817,-81.937,436.891,171.369,26.397,154.943
C02659=1060.811,-82.220,436.903,171.366,26.396,154.943
C02660=1060.803,-82.502,436.915,171.365,26.394,154.943
C02661=1060.796,-82.785,436.927,171.363,26.393,154.943
C02662=1060.789,-83.066,436.939,171.360,26.391,154.943
C02663=1060.783,-83.316,436.951,171.359,26.390,154.943
C02664=1060.777,-83.566,436.961,171.357,26.388,154.942
C02665=1060.771,-83.815,436.972,171.355,26.387,154.942
C02666=1060.764,-84.065,436.983,171.354,26.385,154.942
C02667=1060.758,-84.315,436.994,171.352,26.384,154.942
C02668=1060.752,-84.565,437.005,171.350,26.383,154.942
C02669=1060.745,-84.814,437.015,171.348,26.381,154.942
C02670=1060.740,-85.064,437.026,171.347,26.380,154.942
C02671=1060.733,-85.314,437.038,171.345,26.379,154.942
C02672=1060.727,-85.563,437.048,171.343,26.377,154.942
C02673=1060.721,-85.813,437.059,171.342,26.376,154.942
C02674=1060.715,-86.063,437.070,171.340,26.374,154.942
C02675=1060.709,-86.313,437.079,171.338,26.373,154.942
C02676=1060.702,-86.563,437.091,171.336,26.371,154.942
C02677=1060.697,-86.812,437.102,171.334,26.370,154.942
C02678=1060.690,-87.061,437.112,171.332,26.369,154.942
C02679=1060.684,-87.312,437.123,171.330,26.368,154.942
C02680=1060.678,-87.561,437.134,171.329,26.366,154.942
C02681=1060.672,-87.810,437.144,171.327,26.365,154.942
C02682=1060.665,-88.060,437.156,171.325,26.364,154.942
C02683=1060.659,-88.310,437.166,171.323,26.363,154.941
C02684=1060.653,-88.560,437.176,171.322,26.361,154.941
C02685=1060.647,-88.810,437.187,171.320,26.360,154.941
C02686=1060.641,-89.059,437.198,171.318,26.359,154.941
C02687=1060.635,-89.309,437.208,171.316,26.357,154.941
C02688=1060.629,-89.558,437.219,171.315,26.356,154.941
C02689=1060.623,-89.808,437.231,171.313,26.354,154.941
C02690=1060.616,-90.058,437.240,171.311,26.353,154.941
C02691=1060.611,-90.308,437.251,171.309,26.352,154.941
C02692=1060.604,-90.558,437.262,171.307,26.350,154.941
C02693=1060.598,-90.807,437.272,171.305,26.349,154.941
C02694=1060.592,-91.056,437.283,171.303,26.348,154.941
C02695=1060.586,-91.306,437.293,171.302,26.347,154.941
C02696=1060.580,-91.556,437.304,171.300,26.345,154.941
C02697=1060.574,-91.806,437.315,171.298,26.344,154.941
C02698=1060.567,-92.055,437.325,171.297,26.343,154.941
C02699=1060.562,-92.305,437.335,171.295,26.341,154.941
C02700=1060.556,-92.555,437.347,171.293,26.340,154.941
C02701=1060.549,-92.805,437.357,171.291,26.339,154.941
C02702=1060.543,-93.054,437.368,171.290,26.338,154.941
C02703=1060.537,-93.304,437.377,171.288,26.336,154.941
C02704=1060.532,-93.553,437.388,171.286,26.335,154.941
C02705=1060.525,-93.804,437.400,171.284,26.334,154.940
C02706=1060.519,-94.053,437.409,171.282,26.332,154.941
C02707=1060.513,-94.303,437.420,171.280,26.331,154.940
C02708=1060.507,-94.552,437.430,171.278,26.330,154.940
C02709=1060.501,-94.803,437.441,171.276,26.329,154.940
C02710=1060.494,-95.052,437.451,171.275,26.328,154.940
C02711=1060.489,-95.301,437.462,171.273,26.326,154.940
C02712=1060.483,-95.552,437.472,171.271,26.325,154.940
C02713=1060.477,-95.801,437.482,171.270,26.324,154.940
C02714=1060.471,-96.050,437.493,171.268,26.323,154.940
C02715=1060.464,-96.301,437.503,171.266,26.321,154.940
C02716=1060.458,-96.550,437.514,171.264,26.320,154.940
C02717=1060.452,-96.800,437.524,171.263,26.319,154.940
C02718=1060.447,-97.050,437.535,171.261,26.318,154.940
C02719=1060.441,-97.299,437.545,171.259,26.317,154.940
C02720=1060.435,-97.549,437.555,171.257,26.316,154.940
C02721=1060.428,-97.799,437.566,171.256,26.314,154.940
C02722=1060.422,-98.049,437.576,171.253,26.313,154.940
C02723=1060.415,-98.333,437.587,171.251,26.312,154.940
C02724=1060.408,-98.618,437.599,171.249,26.311,154.940
C02725=1060.401,-98.902,437.611,171.247,26.309,154.940
C02726=1060.394,-99.187,437.622,171.245,26.308,154.940
C02727=1060.388,-99.436,437.633,171.243,26.307,154.940
C02728=1060.382,-99.686,437.643,171.241,26.306,154.940
C02729=1060.375,-99.936,437.653,171.240,26.305,154.940
C02730=1060.369,-100.186,437.664,171.238,26.303,154.940
C02731=1060.363,-100.435,437.674,171.236,26.302,154.940
C02732=1060.357,-100.685,437.683,171.234,26.302,154.940
C02733=1060.351,-100.935,437.694,171.233,26.300,154.940
C02734=1060.345,-101.184,437.704,171.230,26.299,154.940
C02735=1060.339,-101.434,437.713,171.228,26.298,154.940
C02736=1060.332,-101.684,437.725,171.226,26.297,154.940
C02737=1060.326,-101.934,437.734,171.225,26.296,154.940
C02738=1060.320,-102.183,437.745,171.223,26.294,154.940
C02739=1060.314,-102.433,437.755,171.221,26.294,154.940
C02740=1060.308,-102.683,437.765,171.219,26.293,154.940
C02741=1060.301,-102.932,437.775,171.217,26.292,154.940
C02742=1060.296,-103.182,437.785,171.216,26.290,154.940
C02743=1060.290,-103.432,437.795,171.214,26.289,154.940
C02744=1060.283,-103.681,437.805,171.212,26.289,154.940
C02745=1060.277,-103.932,437.816,171.210,26.287,154.940
C02746=1060.271,-104.181,437.825,171.209,26.286,154.940
C02747=1060.265,-104.431,437.835,171.207,26.285,154.940
C02748=1060.258,-104.680,437.845,171.205,26.285,154.940
C02749=1060.253,-104.931,437.855,171.202,26.283,154.940
C02750=1060.247,-105.180,437.865,171.201,26.282,154.940
C02751=1060.240,-105.429,437.875,171.199,26.281,154.940
C02752=1060.234,-105.679,437.885,171.197,26.280,154.940
C02753=1060.229,-105.929,437.895,171.195,26.279,154.940
C02754=1060.222,-106.179,437.905,171.193,26.278,154.940
C02755=1060.216,-106.428,437.915,171.192,26.277,154.940
C02756=1060.210,-106.678,437.924,171.190,26.276,154.940
C02757=1060.204,-106.928,437.935,171.188,26.275,154.940
C02758=1060.198,-107.177,437.945,171.186,26.274,154.940
C02759=1060.192,-107.427,437.954,171.184,26.273,154.940
C02760=1060.185,-107.677,437.964,171.183,26.272,154.940
C02761=1060.178,-107.927,437.975,171.181,26.271,154.940
C02762=1060.173,-108.177,437.985,171.179,26.270,154.940
C02763=1060.167,-108.427,437.994,171.176,26.269,154.940
C02764=1060.161,-108.677,438.004,171.174,26.268,154.941
C02765=1060.154,-108.926,438.014,171.173,26.267,154.941
C02766=1060.148,-109.176,438.024,171.171,26.266,154.941
C02767=1060.142,-109.425,438.033,171.169,26.265,154.941
C02768=1060.136,-109.675,438.043,171.167,26.264,154.941
C02769=1060.129,-109.925,438.052,171.165,26.264,154.941
C02770=1060.124,-110.174,438.063,171.164,26.263,154.941
C02771=1060.118,-110.424,438.073,171.162,26.262,154.941
C02772=1060.111,-110.674,438.083,171.160,26.261,154.941
C02773=1060.105,-110.924,438.092,171.158,26.260,154.941
C02774=1060.099,-111.174,438.102,171.156,26.259,154.941
C02775=1060.093,-111.423,438.111,171.155,26.259,154.941
C02776=1060.086,-111.673,438.121,171.153,26.257,154.941
C02777=1060.080,-111.922,438.131,171.151,26.256,154.941
C02778=1060.074,-112.172,438.141,171.148,26.255,154.941
C02779=1060.068,-112.422,438.150,171.147,26.254,154.941
C02780=1060.062,-112.672,438.160,171.145,26.254,154.941
C02781=1060.056,-112.922,438.170,171.143,26.252,154.941
C02782=1060.050,-113.172,438.179,171.141,26.252,154.941
C02783=1060.044,-113.422,438.189,171.139,26.251,154.941
C02784=1060.038,-113.671,438.199,171.137,26.250,154.941
C02785=1060.031,-113.921,438.209,171.136,26.250,154.941
C02786=1060.025,-114.170,438.218,171.134,26.248,154.941
C02787=1060.019,-114.453,438.229,171.132,26.248,154.941
C02788=1060.011,-114.737,438.239,171.129,26.246,154.942
C02789=1060.005,-115.019,438.251,171.127,26.246,154.942
C02790=1059.998,-115.302,438.262,171.126,26.245,154.942
C02791=1059.992,-115.552,438.271,171.124,26.244,154.942
C02792=1059.985,-115.802,438.281,171.121,26.243,154.942
C02793=1059.979,-116.052,438.290,171.119,26.242,154.942
C02794=1059.972,-116.301,438.299,171.117,26.241,154.942
C02795=1059.966,-116.551,438.309,171.116,26.240,154.942
C02796=1059.961,-116.800,438.318,171.114,26.240,154.942
C02797=1059.954,-117.050,438.328,171.112,26.239,154.942
C02798=1059.948,-117.300,438.337,171.110,26.238,154.942
C02799=1059.942,-117.550,438.347,171.108,26.237,154.942
C02800=1059.936,-117.799,438.356,171.106,26.237,154.942
C02801=1059.930,-118.049,438.366,171.105,26.236,154.942
C02802=1059.924,-118.299,438.376,171.103,26.235,154.942
C02803=1059.917,-118.549,438.385,171.101,26.235,154.942
C02804=1059.911,-118.799,438.395,171.099,26.234,154.943
C02805=1059.905,-119.048,438.404,171.097,26.233,154.943
C02806=1059.899,-119.298,438.414,171.095,26.232,154.943
C02807=1059.894,-119.548,438.422,171.093,26.232,154.943
C02808=1059.887,-119.798,438.432,171.091,26.231,154.943
C02809=1059.881,-120.047,438.441,171.089,26.230,154.943
C02810=1059.874,-120.297,438.450,171.087,26.229,154.943
C02811=1059.868,-120.547,438.460,171.085,26.228,154.943
C02812=1059.862,-120.797,438.470,171.083,26.228,154.943
C02813=1059.856,-121.046,438.479,171.082,26.227,154.943
C02814=1059.850,-121.295,438.488,171.080,26.226,154.943
C02815=1059.844,-121.546,438.497,171.078,26.226,154.943
C02816=1059.838,-121.796,438.507,171.076,26.225,154.943
C02817=1059.831,-122.045,438.516,171.074,26.224,154.944
C02818=1059.825,-122.295,438.525,171.072,26.223,154.944
C02819=1059.819,-122.545,438.535,171.070,26.223,154.944
C02820=1059.813,-122.795,438.544,171.069,26.222,154.944
C02821=1059.808,-123.044,438.553,171.067,26.222,154.944
C02822=1059.801,-123.294,438.562,171.065,26.221,154.944
C02823=1059.794,-123.544,438.571,171.063,26.220,154.944
C02824=1059.788,-123.793,438.581,171.060,26.220,154.944
C02825=1059.782,-124.044,438.590,171.058,26.218,154.944
C02826=1059.777,-124.293,438.599,171.057,26.218,154.944
C02827=1059.771,-124.543,438.609,171.055,26.217,154.944
C02828=1059.764,-124.792,438.618,171.053,26.217,154.944
C02829=1059.758,-125.043,438.626,171.051,26.216,154.945
C02830=1059.752,-125.292,438.636,171.049,26.216,154.945
C02831=1059.746,-125.542,438.646,171.047,26.215,154.945
C02832=1059.739,-125.791,438.654,171.045,26.214,154.945
C02833=1059.733,-126.041,438.663,171.043,26.214,154.945
C02834=1059.727,-126.291,438.673,171.042,26.213,154.945
C02835=1059.721,-126.541,438.682,171.040,26.213,154.945
C02836=1059.714,-126.791,438.690,171.038,26.212,154.945
C02837=1059.709,-127.040,438.700,171.036,26.212,154.945
C02838=1059.703,-127.290,438.709,171.034,26.211,154.945
C02839=1059.696,-127.540,438.717,171.032,26.210,154.946
C02840=1059.690,-127.790,438.727,171.030,26.210,154.946
C02841=1059.685,-128.039,438.737,171.028,26.208,154.946
C02842=1059.681,-128.290,438.747,171.027,26.207,154.946
C02843=1059.679,-128.540,438.758,171.025,26.205,154.945
C02844=1059.677,-128.791,438.770,171.024,26.203,154.945
C02845=1059.677,-129.041,438.782,171.023,26.199,154.945
C02846=1059.679,-129.291,438.795,171.021,26.196,154.944
C02847=1059.681,-129.543,438.809,171.020,26.191,154.943
C02848=1059.686,-129.794,438.823,171.020,26.186,154.943
C02849=1059.692,-130.045,438.839,171.019,26.181,154.942
C02850=1059.699,-130.296,438.855,171.020,26.174,154.941
C02851=1059.321,-130.318,438.658,170.972,26.334,154.974
C02852=1059.314,-130.069,438.642,170.972,26.340,154.975
C02853=1059.309,-129.818,438.627,170.972,26.346,154.976
C02854=1059.303,-129.567,438.612,170.973,26.351,154.977
C02855=1059.301,-129.314,438.598,170.974,26.355,154.977
C02856=1059.299,-129.064,438.585,170.975,26.359,154.978
C02857=1059.299,-128.814,438.574,170.976,26.362,154.978
C02858=1059.300,-128.563,438.561,170.978,26.365,154.979
C02859=1059.303,-128.312,438.551,170.979,26.367,154.979
C02860=1059.306,-128.062,438.540,170.981,26.368,154.979
C02861=1059.312,-127.813,438.531,170.983,26.369,154.979
C02862=1059.318,-127.563,438.522,170.984,26.370,154.979
C02863=1059.324,-127.313,438.512,170.986,26.371,154.979
C02864=1059.330,-127.063,438.503,170.988,26.371,154.979
C02865=1059.336,-126.814,438.495,170.990,26.372,154.979
C02866=1059.342,-126.564,438.485,170.992,26.372,154.978
C02867=1059.348,-126.314,438.476,170.994,26.373,154.978
C02868=1059.355,-126.064,438.467,170.996,26.373,154.978
C02869=1059.361,-125.814,438.458,170.998,26.374,154.978
C02870=1059.367,-125.565,438.448,170.999,26.374,154.978
C02871=1059.373,-125.315,438.440,171.001,26.375,154.978
C02872=1059.380,-125.065,438.431,171.003,26.376,154.978
C02873=1059.386,-124.816,438.421,171.005,26.376,154.978
C02874=1059.392,-124.566,438.411,171.007,26.377,154.978
C02875=1059.398,-124.315,438.403,171.009,26.377,154.978
C02876=1059.404,-124.067,438.394,171.012,26.378,154.977
C02877=1059.410,-123.817,438.384,171.013,26.379,154.977
C02878=1059.416,-123.567,438.375,171.015,26.380,154.977
C02879=1059.422,-123.316,438.366,171.017,26.380,154.977
C02880=1059.429,-123.067,438.356,171.019,26.381,154.977
C02881=1059.434,-122.818,438.347,171.021,26.382,154.977
C02882=1059.441,-122.568,438.338,171.023,26.382,154.977
C02883=1059.447,-122.318,438.329,171.025,26.383,154.977
C02884=1059.453,-122.068,438.320,171.026,26.383,154.977
C02885=1059.459,-121.818,438.310,171.028,26.384,154.977
C02886=1059.465,-121.568,438.301,171.030,26.385,154.977
C02887=1059.471,-121.319,438.292,171.032,26.386,154.977
C02888=1059.477,-121.069,438.282,171.034,26.386,154.976
C02889=1059.484,-120.820,438.273,171.036,26.387,154.976
C02890=1059.490,-120.570,438.264,171.037,26.388,154.976
C02891=1059.496,-120.320,438.255,171.040,26.389,154.976
C02892=1059.502,-120.070,438.245,171.042,26.389,154.976
C02893=1059.508,-119.820,438.235,171.044,26.390,154.976
C02894=1059.515,-119.570,438.226,171.046,26.391,154.976
C02895=1059.520,-119.321,438.217,171.048,26.391,154.976
C02896=1059.526,-119.071,438.207,171.049,26.392,154.976
C02897=1059.533,-118.822,438.198,171.051,26.393,154.976
C02898=1059.539,-118.572,438.188,171.053,26.394,154.976
C02899=1059.546,-118.322,438.179,171.055,26.394,154.976
C02900=1059.552,-118.073,438.169,171.057,26.395,154.976
C02901=1059.558,-117.823,438.160,171.059,26.395,154.975
C02902=1059.564,-117.572,438.151,171.060,26.397,154.975
C02903=1059.570,-117.323,438.141,171.062,26.397,154.975
C02904=1059.576,-117.073,438.132,171.064,26.398,154.975
C02905=1059.582,-116.824,438.123,171.067,26.399,154.975
C02906=1059.588,-116.574,438.113,171.069,26.400,154.975
C02907=1059.594,-116.324,438.104,171.071,26.400,154.975
C02908=1059.600,-116.074,438.094,171.072,26.401,154.975
C02909=1059.606,-115.824,438.084,171.074,26.402,154.975
C02910=1059.613,-115.575,438.075,171.076,26.403,154.975
C02911=1059.619,-115.325,438.065,171.078,26.404,154.975
C02912=1059.626,-115.042,438.054,171.080,26.404,154.975
C02913=1059.633,-114.759,438.044,171.083,26.406,154.975
C02914=1059.640,-114.476,438.033,171.084,26.406,154.975
C02915=1059.647,-114.193,438.021,171.086,26.407,154.975
C02916=1059.653,-113.943,438.011,171.088,26.408,154.975
C02917=1059.659,-113.693,438.002,171.090,26.409,154.974
C02918=1059.665,-113.443,437.992,171.093,26.410,154.974
C02919=1059.671,-113.194,437.983,171.094,26.411,154.974
C02920=1059.677,-112.944,437.973,171.096,26.412,154.974
C02921=1059.683,-112.695,437.964,171.098,26.412,154.974
C02922=1059.690,-112.445,437.954,171.100,26.413,154.974
C02923=1059.696,-112.195,437.945,171.102,26.414,154.974
C02924=1059.702,-111.946,437.934,171.103,26.415,154.974
C02925=1059.708,-111.696,437.925,171.105,26.416,154.974
C02926=1059.714,-111.446,437.915,171.107,26.417,154.974
C02927=1059.720,-111.196,437.905,171.109,26.417,154.974
C02928=1059.726,-110.946,437.896,171.111,26.419,154.974
C02929=1059.732,-110.697,437.886,171.113,26.419,154.974
C02930=1059.739,-110.447,437.876,171.114,26.420,154.974
C02931=1059.745,-110.198,437.866,171.116,26.421,154.974
C02932=1059.751,-109.948,437.857,171.119,26.422,154.974
C02933=1059.757,-109.698,437.847,171.121,26.423,154.974
C02934=1059.763,-109.448,437.837,171.123,26.424,154.974
C02935=1059.769,-109.198,437.827,171.124,26.425,154.974
C02936=1059.775,-108.949,437.817,171.126,26.426,154.974
C02937=1059.782,-108.698,437.807,171.128,26.427,154.974
C02938=1059.788,-108.449,437.798,171.130,26.427,154.974
C02939=1059.795,-108.199,437.788,171.132,26.429,154.974
C02940=1059.801,-107.950,437.778,171.133,26.430,154.974
C02941=1059.807,-107.700,437.768,171.135,26.430,154.974
C02942=1059.813,-107.450,437.759,171.137,26.432,154.974
C02943=1059.819,-107.200,437.748,171.139,26.433,154.974
C02944=1059.825,-106.951,437.738,171.141,26.433,154.973
C02945=1059.831,-106.701,437.729,171.143,26.435,154.973
C02946=1059.838,-106.451,437.719,171.145,26.436,154.973
C02947=1059.843,-106.202,437.708,171.147,26.436,154.973
C02948=1059.850,-105.952,437.699,171.149,26.438,154.973
C02949=1059.856,-105.702,437.689,171.150,26.439,154.973
C02950=1059.862,-105.453,437.679,171.152,26.439,154.973
C02951=1059.868,-105.203,437.669,171.154,26.440,154.973
C02952=1059.874,-104.953,437.659,171.156,26.442,154.973
C02953=1059.880,-104.704,437.649,171.158,26.443,154.973
C02954=1059.886,-104.453,437.638,171.159,26.443,154.973
C02955=1059.892,-104.203,437.629,171.161,26.444,154.973
C02956=1059.899,-103.954,437.618,171.163,26.446,154.973
C02957=1059.905,-103.704,437.609,171.165,26.447,154.973
C02958=1059.911,-103.454,437.599,171.167,26.447,154.973
C02959=1059.917,-103.205,437.588,171.169,26.449,154.973
C02960=1059.923,-102.955,437.579,171.171,26.450,154.973
C02961=1059.929,-102.706,437.568,171.173,26.451,154.973
C02962=1059.935,-102.456,437.558,171.175,26.452,154.973
C02963=1059.942,-102.207,437.548,171.176,26.453,154.973
C02964=1059.948,-101.956,437.537,171.178,26.454,154.973
C02965=1059.954,-101.706,437.528,171.180,26.455,154.973
C02966=1059.960,-101.457,437.518,171.182,26.456,154.973
C02967=1059.966,-101.207,437.507,171.183,26.457,154.973
C02968=1059.972,-100.958,437.497,171.185,26.459,154.973
C02969=1059.978,-100.708,437.488,171.187,26.459,154.973
C02970=1059.984,-100.458,437.477,171.189,26.460,154.973
C02971=1059.991,-100.208,437.467,171.191,26.461,154.973
C02972=1059.997,-99.959,437.456,171.192,26.463,154.973
C02973=1060.003,-99.708,437.446,171.195,26.464,154.973
C02974=1060.009,-99.459,437.436,171.197,26.465,154.973
C02975=1060.015,-99.209,437.426,171.199,26.466,154.973
C02976=1060.022,-98.925,437.415,171.200,26.467,154.973
C02977=1060.029,-98.640,437.403,171.202,26.469,154.973
C02978=1060.037,-98.355,437.391,171.205,26.470,154.973
C02979=1060.044,-98.071,437.379,171.207,26.471,154.973
C02980=1060.050,-97.821,437.369,171.208,26.472,154.973
C02981=1060.056,-97.571,437.359,171.210,26.473,154.973
C02982=1060.062,-97.321,437.349,171.212,26.475,154.973
C02983=1060.067,-97.072,437.338,171.214,26.476,154.973
C02984=1060.075,-96.822,437.327,171.215,26.477,154.973
C02985=1060.080,-96.572,437.317,171.218,26.478,154.973
C02986=1060.086,-96.323,437.307,171.220,26.480,154.973
C02987=1060.092,-96.073,437.296,171.222,26.481,154.973
C02988=1060.098,-95.823,437.286,171.223,26.482,154.973
C02989=1060.104,-95.574,437.276,171.225,26.483,154.973
C02990=1060.110,-95.323,437.265,171.227,26.484,154.973
C02991=1060.117,-95.074,437.255,171.229,26.485,154.973
C02992=1060.122,-94.825,437.244,171.230,26.486,154.973
C02993=1060.129,-94.575,437.234,171.232,26.488,154.974
C02994=1060.134,-94.325,437.224,171.234,26.489,154.974
C02995=1060.141,-94.075,437.212,171.236,26.490,154.974
C02996=1060.147,-93.825,437.203,171.237,26.492,154.974
C02997=1060.153,-93.576,437.192,171.239,26.493,154.974
C02998=1060.159,-93.327,437.182,171.241,26.494,154.974
C02999=1060.165,-93.077,437.171,171.244,26.495,154.974
C03000=1060.171,-92.826,437.160,171.245,26.497,154.974
C03001=1060.177,-92.577,437.150,171.247,26.498,154.974
C03002=1060.183,-92.328,437.139,171.249,26.499,154.974
C03003=1060.189,-92.078,437.129,171.250,26.501,154.974
C03004=1060.196,-91.828,437.118,171.252,26.502,154.974
C03005=1060.201,-91.578,437.107,171.254,26.503,154.974
C03006=1060.208,-91.329,437.097,171.256,26.504,154.974
C03007=1060.213,-91.079,437.086,171.257,26.506,154.974
C03008=1060.219,-90.829,437.076,171.259,26.507,154.974
C03009=1060.226,-90.579,437.065,171.261,26.508,154.974
C03010=1060.232,-90.330,437.054,171.263,26.509,154.974
C03011=1060.239,-90.080,437.044,171.264,26.510,154.974
C03012=1060.245,-89.831,437.033,171.266,26.512,154.974
C03013=1060.250,-89.581,437.023,171.268,26.513,154.974
C03014=1060.256,-89.331,437.012,171.270,26.515,154.974
C03015=1060.263,-89.081,437.001,171.272,26.516,154.974
C03016=1060.269,-88.832,436.990,171.274,26.517,154.974
C03017=1060.275,-88.582,436.980,171.276,26.519,154.975
C03018=1060.281,-88.332,436.969,171.277,26.520,154.975
C03019=1060.287,-88.082,436.959,171.279,26.521,154.975
C03020=1060.293,-87.833,436.948,171.281,26.522,154.975
C03021=1060.300,-87.583,436.937,171.283,26.524,154.975
C03022=1060.305,-87.333,436.926,171.284,26.525,154.975
C03023=1060.312,-87.084,436.916,171.286,26.526,154.975
C03024=1060.318,-86.834,436.905,171.288,26.528,154.975
C03025=1060.324,-86.584,436.894,171.290,26.529,154.975
C03026=1060.330,-86.335,436.884,171.291,26.530,154.975
C03027=1060.337,-86.085,436.872,171.293,26.531,154.975
C03028=1060.342,-85.836,436.861,171.295,26.533,154.975
C03029=1060.349,-85.586,436.851,171.297,26.535,154.975
C03030=1060.355,-85.336,436.841,171.299,26.536,154.975
C03031=1060.361,-85.086,436.830,171.301,26.537,154.975
C03032=1060.368,-84.836,436.819,171.303,26.539,154.975
C03033=1060.374,-84.587,436.808,171.304,26.540,154.975
C03034=1060.379,-84.337,436.797,171.306,26.541,154.975
C03035=1060.386,-84.087,436.787,171.308,26.543,154.975
C03036=1060.392,-83.838,436.776,171.309,26.544,154.975
C03037=1060.398,-83.588,436.765,171.311,26.546,154.976
C03038=1060.404,-83.338,436.754,171.313,26.547,154.976
C03039=1060.411,-83.089,436.743,171.315,26.548,154.976
C03040=1060.417,-82.806,436.730,171.317,26.550,154.976
C03041=1060.425,-82.524,436.718,171.319,26.551,154.976
C03042=1060.432,-82.242,436.706,171.321,26.553,154.976
C03043=1060.438,-81.959,436.694,171.323,26.554,154.976
C03044=1060.446,-81.710,436.682,171.325,26.556,154.976
C03045=1060.451,-81.460,436.671,171.327,26.557,154.976
C03046=1060.458,-81.210,436.660,171.328,26.559,154.976
C03047=1060.464,-80.961,436.650,171.330,26.560,154.976
C03048=1060.470,-80.711,436.639,171.332,26.561,154.976
C03049=1060.476,-80.461,436.628,171.334,26.563,154.976
C03050=1060.483,-80.211,436.617,171.335,26.564,154.976
C03051=1060.489,-79.962,436.606,171.337,26.566,154.977
C03052=1060.495,-79.712,436.595,171.339,26.567,154.977
C03053=1060.501,-79.462,436.584,171.340,26.569,154.977
C03054=1060.507,-79.213,436.573,171.342,26.570,154.977
C03055=1060.513,-78.963,436.561,171.344,26.571,154.977
C03056=1060.519,-78.714,436.550,171.346,26.573,154.977
C03057=1060.526,-78.463,436.539,171.348,26.575,154.977
C03058=1060.531,-78.214,436.528,171.350,26.576,154.977
C03059=1060.538,-77.964,436.517,171.352,26.578,154.977
C03060=1060.544,-77.715,436.506,171.353,26.579,154.977
C03061=1060.549,-77.465,436.495,171.355,26.580,154.977
C03062=1060.556,-77.215,436.483,171.357,26.582,154.977
C03063=1060.562,-76.966,436.473,171.358,26.583,154.977
C03064=1060.569,-76.716,436.462,171.360,26.585,154.978
C03065=1060.575,-76.467,436.450,171.362,26.586,154.978
C03066=1060.581,-76.217,436.439,171.363,26.588,154.978
C03067=1060.587,-75.967,436.428,171.365,26.590,154.978
C03068=1060.593,-75.717,436.417,171.367,26.591,154.978
C03069=1060.599,-75.468,436.405,171.368,26.593,154.978
C03070=1060.605,-75.218,436.394,171.370,26.594,154.978
C03071=1060.611,-74.969,436.383,171.372,26.595,154.978
C03072=1060.618,-74.718,436.372,171.374,26.597,154.978
C03073=1060.624,-74.469,436.360,171.375,26.598,154.978
C03074=1060.630,-74.219,436.349,171.378,26.600,154.979
C03075=1060.636,-73.970,436.338,171.380,26.602,154.979
C03076=1060.642,-73.720,436.326,171.381,26.603,154.979
C03077=1060.647,-73.470,436.315,171.383,26.605,154.979
C03078=1060.654,-73.220,436.304,171.385,26.607,154.979
C03079=1060.660,-72.971,436.292,171.386,26.608,154.979
C03080=1060.666,-72.721,436.281,171.388,26.610,154.979
C03081=1060.672,-72.472,436.270,171.390,26.611,154.979
C03082=1060.678,-72.222,436.257,171.391,26.613,154.979
C03083=1060.683,-71.972,436.246,171.393,26.615,154.980
C03084=1060.690,-71.723,436.234,171.395,26.616,154.980
C03085=1060.696,-71.473,436.224,171.396,26.618,154.980
C03086=1060.702,-71.223,436.212,171.398,26.620,154.980
C03087=1060.707,-70.974,436.200,171.400,26.621,154.980
C03088=1060.714,-70.724,436.189,171.401,26.623,154.980
C03089=1060.720,-70.475,436.177,171.403,26.625,154.980
C03090=1060.726,-70.225,436.166,171.405,26.626,154.980
C03091=1060.732,-69.975,436.155,171.406,26.628,154.981
C03092=1060.738,-69.725,436.143,171.408,26.630,154.981
C03093=1060.744,-69.476,436.132,171.410,26.631,154.981
C03094=1060.750,-69.226,436.120,171.412,26.633,154.981
C03095=1060.757,-68.976,436.109,171.414,26.635,154.981
C03096=1060.762,-68.727,436.096,171.416,26.636,154.981
C03097=1060.768,-68.477,436.085,171.417,26.638,154.981
C03098=1060.774,-68.228,436.074,171.419,26.640,154.981
C03099=1060.781,-67.978,436.062,171.421,26.642,154.982
C03100=1060.786,-67.728,436.050,171.422,26.643,154.982
C03101=1060.792,-67.478,436.039,171.424,26.645,154.982
C03102=1060.799,-67.229,436.027,171.426,26.647,154.982
C03103=1060.805,-66.979,436.016,171.427,26.648,154.982
C03104=1060.811,-66.699,436.002,171.429,26.650,154.982
C03105=1060.818,-66.419,435.989,171.431,26.652,154.982
C03106=1060.825,-66.138,435.976,171.433,26.654,154.982
C03107=1060.832,-65.859,435.963,171.435,26.656,154.983
C03108=1060.838,-65.609,435.952,171.436,26.657,154.983
C03109=1060.844,-65.359,435.940,171.438,26.659,154.983
C03110=1060.850,-65.110,435.928,171.440,26.661,154.983
C03111=1060.856,-64.860,435.917,171.441,26.663,154.983
C03112=1060.862,-64.610,435.905,171.443,26.664,154.983
C03113=1060.868,-64.360,435.893,171.445,26.666,154.983
C03114=1060.875,-64.111,435.881,171.446,26.668,154.984
C03115=1060.881,-63.862,435.870,171.448,26.669,154.984
C03116=1060.886,-63.611,435.858,171.451,26.671,154.984
C03117=1060.893,-63.362,435.846,171.452,26.673,154.984
C03118=1060.899,-63.113,435.834,171.454,26.675,154.984
C03119=1060.905,-62.862,435.823,171.456,26.677,154.984
C03120=1060.911,-62.613,435.811,171.457,26.678,154.984
C03121=1060.917,-62.364,435.799,171.459,26.680,154.985
C03122=1060.923,-62.113,435.787,171.460,26.682,154.985
C03123=1060.930,-61.864,435.775,171.462,26.684,154.985
C03124=1060.936,-61.615,435.764,171.464,26.685,154.985
C03125=1060.942,-61.365,435.752,171.465,26.687,154.985
C03126=1060.948,-61.115,435.740,171.467,26.689,154.985
C03127=1060.954,-60.865,435.728,171.469,26.691,154.985
C03128=1060.961,-60.616,435.716,171.470,26.692,154.986
C03129=1060.966,-60.366,435.704,171.472,26.694,154.986
C03130=1060.973,-60.116,435.692,171.474,26.696,154.986
C03131=1060.979,-59.868,435.681,171.475,26.697,154.986
C03132=1060.985,-59.618,435.668,171.477,26.699,154.986
C03133=1060.991,-59.367,435.657,171.479,26.701,154.986
C03134=1060.998,-59.118,435.645,171.480,26.703,154.986
C03135=1061.003,-58.869,435.633,171.482,26.704,154.987
C03136=1061.010,-58.619,435.621,171.484,26.706,154.987
C03137=1061.016,-58.369,435.610,171.485,26.708,154.987
C03138=1061.022,-58.119,435.597,171.487,26.710,154.987
C03139=1061.028,-57.870,435.586,171.489,26.711,154.987
C03140=1061.034,-57.620,435.573,171.491,26.713,154.987
C03141=1061.041,-57.371,435.561,171.493,26.715,154.987
C03142=1061.047,-57.121,435.549,171.495,26.717,154.988
C03143=1061.053,-56.871,435.537,171.496,26.718,154.988
C03144=1061.059,-56.622,435.526,171.498,26.720,154.988
C03145=1061.065,-56.372,435.514,171.499,26.722,154.988
C03146=1061.071,-56.122,435.501,171.501,26.724,154.988
C03147=1061.078,-55.873,435.489,171.503,26.726,154.988
C03148=1061.085,-55.623,435.477,171.504,26.728,154.989
C03149=1061.090,-55.374,435.465,171.506,26.729,154.989
C03150=1061.097,-55.124,435.453,171.508,26.731,154.989
C03151=1061.102,-54.874,435.441,171.509,26.733,154.989
C03152=1061.109,-54.624,435.429,171.511,26.735,154.989
C03153=1061.116,-54.375,435.417,171.513,26.736,154.989
C03154=1061.121,-54.125,435.405,171.514,26.738,154.989
C03155=1061.127,-53.876,435.393,171.516,26.740,154.990
C03156=1061.133,-53.626,435.381,171.517,26.742,154.990
C03157=1061.140,-53.377,435.369,171.519,26.744,154.990
C03158=1061.147,-53.127,435.357,171.521,26.745,154.990
C03159=1061.153,-52.877,435.344,171.522,26.747,154.990
C03160=1061.159,-52.628,435.332,171.524,26.749,154.990
C03161=1061.165,-52.378,435.320,171.526,26.751,154.991
C03162=1061.171,-52.129,435.308,171.527,26.752,154.991
C03163=1061.178,-51.879,435.296,171.529,26.755,154.991
C03164=1061.184,-51.629,435.284,171.531,26.756,154.991
C03165=1061.190,-51.380,435.272,171.532,26.758,154.991
C03166=1061.196,-51.130,435.259,171.534,26.760,154.991
C03167=1061.203,-50.880,435.247,171.536,26.762,154.991
C03168=1061.210,-50.601,435.233,171.538,26.764,154.992
C03169=1061.217,-50.323,435.220,171.540,26.766,154.992
C03170=1061.224,-50.044,435.206,171.541,26.768,154.992
C03171=1061.230,-49.764,435.192,171.543,26.770,154.992
C03172=1061.236,-49.516,435.180,171.545,26.772,154.992
C03173=1061.242,-49.266,435.167,171.547,26.774,154.993
C03174=1061.248,-49.016,435.155,171.549,26.777,154.993
C03175=1061.254,-48.766,435.142,171.550,26.778,154.993
C03176=1061.261,-48.516,435.130,171.552,26.780,154.993
C03177=1061.267,-48.266,435.118,171.554,26.782,154.993
C03178=1061.273,-48.017,435.105,171.555,26.784,154.994
C03179=1061.279,-47.768,435.093,171.557,26.786,154.994
C03180=1061.285,-47.518,435.080,171.558,26.788,154.994
C03181=1061.291,-47.269,435.068,171.560,26.790,154.994
C03182=1061.297,-47.019,435.055,171.562,26.792,154.994
C03183=1061.303,-46.769,435.043,171.563,26.794,154.995
C03184=1061.309,-46.519,435.031,171.565,26.795,154.995
C03185=1061.316,-46.270,435.018,171.566,26.798,154.995
C03186=1061.321,-46.020,435.005,171.568,26.800,154.995
C03187=1061.327,-45.771,434.993,171.570,26.802,154.995
C03188=1061.333,-45.521,434.981,171.571,26.804,154.996
C03189=1061.339,-45.271,434.968,171.573,26.806,154.996
C03190=1061.345,-45.022,434.955,171.575,26.808,154.996
C03191=1061.352,-44.773,434.943,171.576,26.809,154.996
C03192=1061.358,-44.523,434.930,171.578,26.812,154.996
C03193=1061.364,-44.273,434.918,171.579,26.813,154.996
C03194=1061.370,-44.024,434.905,171.581,26.816,154.997
C03195=1061.377,-43.774,434.893,171.583,26.817,154.997
C03196=1061.383,-43.524,434.880,171.584,26.820,154.997
C03197=1061.389,-43.274,434.868,171.586,26.821,154.997
C03198=1061.395,-43.025,434.854,171.587,26.824,154.998
C03199=1061.401,-42.775,434.842,171.589,26.825,154.998
C03200=1061.407,-42.526,434.830,171.591,26.827,154.998
C03201=1061.414,-42.276,434.817,171.592,26.829,154.998
C03202=1061.420,-42.026,434.804,171.594,26.831,154.998
C03203=1061.425,-41.777,434.791,171.595,26.833,154.999
C03204=1061.432,-41.528,434.779,171.597,26.835,154.999
C03205=1061.438,-41.278,434.766,171.599,26.837,154.999
C03206=1061.444,-41.028,434.754,171.600,26.839,154.999
C03207=1061.450,-40.779,434.740,171.602,26.841,154.999
C03208=1061.456,-40.529,434.728,171.604,26.843,154.999
C03209=1061.463,-40.279,434.716,171.605,26.845,155.000
C03210=1061.469,-40.030,434.703,171.607,26.847,155.000
C03211=1061.475,-39.780,434.690,171.608,26.850,155.000
C03212=1061.481,-39.530,434.677,171.610,26.851,155.000
C03213=1061.487,-39.281,434.664,171.612,26.854,155.001
C03214=1061.494,-39.031,434.652,171.613,26.855,155.001
C03215=1061.500,-38.782,434.639,171.615,26.858,155.001
C03216=1061.506,-38.532,434.626,171.616,26.859,155.001
C03217=1061.512,-38.283,434.613,171.618,26.862,155.001
C03218=1061.518,-38.033,434.601,171.620,26.864,155.002
C03219=1061.524,-37.783,434.588,171.621,26.866,155.002
C03220=1061.530,-37.534,434.575,171.623,26.868,155.002
C03221=1061.536,-37.284,434.562,171.624,26.870,155.002
C03222=1061.542,-37.035,434.549,171.626,26.872,155.002
C03223=1061.548,-36.785,434.536,171.628,26.874,155.003
C03224=1061.554,-36.535,434.523,171.629,26.876,155.003
C03225=1061.560,-36.286,434.511,171.631,26.878,155.003
C03226=1061.567,-36.036,434.497,171.632,26.881,155.003
C03227=1061.573,-35.786,434.485,171.634,26.882,155.004
C03228=1061.579,-35.537,434.471,171.636,26.885,155.004
C03229=1061.585,-35.287,434.459,171.637,26.887,155.004
C03230=1061.591,-35.038,434.446,171.639,26.889,155.004
C03231=1061.597,-34.789,434.432,171.640,26.891,155.004
C03232=1061.604,-34.509,434.418,171.642,26.893,155.005
C03233=1061.610,-34.232,434.404,171.643,26.895,155.005
C03234=1061.617,-33.953,434.389,171.646,26.898,155.005
C03235=1061.624,-33.674,434.374,171.647,26.900,155.006
C03236=1061.630,-33.424,434.361,171.649,26.903,155.006
C03237=1061.636,-33.175,434.348,171.651,26.904,155.006
C03238=1061.642,-32.925,434.335,171.652,26.907,155.006
C03239=1061.648,-32.676,434.322,171.654,26.909,155.006
C03240=1061.654,-32.426,434.309,171.655,26.911,155.007
C03241=1061.660,-32.177,434.296,171.657,26.913,155.007
C03242=1061.667,-31.928,434.283,171.659,26.915,155.007
C03243=1061.672,-31.678,434.270,171.660,26.918,155.007
C03244=1061.679,-31.428,434.257,171.662,26.919,155.008
C03245=1061.686,-31.178,434.243,171.663,26.922,155.008
C03246=1061.691,-30.928,434.231,171.665,26.924,155.008
C03247=1061.698,-30.679,434.218,171.667,26.926,155.008
C03248=1061.704,-30.430,434.204,171.668,26.928,155.008
C03249=1061.709,-30.180,434.191,171.670,26.930,155.009
C03250=1061.715,-29.931,434.178,171.671,26.932,155.009
C03251=1061.721,-29.681,434.165,171.673,26.934,155.009
C03252=1061.728,-29.431,434.151,171.675,26.936,155.009
C03253=1061.734,-29.181,434.138,171.676,26.939,155.010
C03254=1061.740,-28.932,434.125,171.678,26.941,155.010
C03255=1061.747,-28.683,434.112,171.679,26.943,155.010
C03256=1061.753,-28.434,434.099,171.681,26.945,155.010
C03257=1061.759,-28.184,434.086,171.682,26.947,155.011
C03258=1061.766,-27.934,434.072,171.684,26.950,155.011
C03259=1061.772,-27.685,434.059,171.686,26.951,155.011
C03260=1061.777,-27.435,434.045,171.687,26.954,155.011
C03261=1061.783,-27.185,434.033,171.689,26.956,155.012
C03262=1061.789,-26.936,434.019,171.690,26.958,155.012
C03263=1061.796,-26.686,434.006,171.691,26.960,155.012
C03264=1061.802,-26.437,433.993,171.693,26.962,155.012
C03265=1061.808,-26.187,433.979,171.694,26.964,155.013
C03266=1061.814,-25.937,433.966,171.696,26.967,155.013
C03267=1061.820,-25.688,433.953,171.697,26.969,155.013
C03268=1061.825,-25.438,433.939,171.699,26.971,155.013
C03269=1061.832,-25.189,433.926,171.700,26.973,155.014
C03270=1061.838,-24.939,433.912,171.702,26.976,155.014
C03271=1061.844,-24.689,433.898,171.704,26.977,155.014
C03272=1061.850,-24.440,433.885,171.705,26.980,155.014
C03273=1061.856,-24.190,433.872,171.707,26.982,155.015
C03274=1061.862,-23.941,433.859,171.708,26.984,155.015
C03275=1061.868,-23.691,433.845,171.710,26.987,155.015
C03276=1061.875,-23.441,433.832,171.712,26.989,155.015
C03277=1061.880,-23.192,433.818,171.713,26.991,155.016
C03278=1061.886,-22.943,433.804,171.715,26.993,155.016
C03279=1061.892,-22.693,433.791,171.716,26.996,155.016
C03280=1061.899,-22.443,433.777,171.718,26.998,155.016
C03281=1061.905,-22.194,433.764,171.719,27.000,155.017
C03282=1061.911,-21.945,433.750,171.721,27.002,155.017
C03283=1061.916,-21.695,433.737,171.723,27.004,155.017
C03284=1061.923,-21.445,433.723,171.724,27.007,155.017
C03285=1061.929,-21.196,433.710,171.726,27.009,155.018
C03286=1061.935,-20.946,433.696,171.727,27.011,155.018
C03287=1061.941,-20.697,433.683,171.729,27.013,155.018
C03288=1061.948,-20.447,433.669,171.730,27.016,155.018
C03289=1061.953,-20.197,433.655,171.732,27.018,155.019
C03290=1061.960,-19.948,433.642,171.734,27.020,155.019
C03291=1061.965,-19.699,433.628,171.735,27.023,155.019
C03292=1061.972,-19.449,433.614,171.737,27.025,155.020
C03293=1061.978,-19.199,433.601,171.738,27.027,155.020
C03294=1061.984,-18.950,433.587,171.740,27.029,155.020
C03295=1061.990,-18.700,433.573,171.740,27.032,155.020
C03296=1061.997,-18.421,433.558,171.743,27.034,155.021
C03297=1062.005,-18.142,433.543,171.745,27.036,155.021
C03298=1062.010,-17.862,433.528,171.746,27.039,155.021
C03299=1062.018,-17.582,433.512,171.748,27.042,155.021
C03300=1062.024,-17.333,433.499,171.749,27.044,155.022
C03301=1062.029,-17.084,433.485,171.751,27.046,155.022
C03302=1062.037,-16.834,433.471,171.752,27.048,155.022
C03303=1062.043,-16.585,433.458,171.754,27.051,155.023
C03304=1062.048,-16.335,433.444,171.755,27.053,155.023
C03305=1062.055,-16.085,433.430,171.757,27.055,155.023
C03306=1062.061,-15.836,433.416,171.759,27.058,155.023
C03307=1062.067,-15.587,433.403,171.760,27.060,155.024
C03308=1062.073,-15.336,433.389,171.762,27.062,155.024
C03309=1062.079,-15.088,433.375,171.763,27.064,155.024
C03310=1062.085,-14.838,433.361,171.765,27.067,155.024
C03311=1062.092,-14.588,433.347,171.766,27.069,155.025
C03312=1062.097,-14.339,433.333,171.768,27.071,155.025
C03313=1062.103,-14.089,433.320,171.769,27.074,155.025
C03314=1062.110,-13.840,433.305,171.771,27.076,155.025
C03315=1062.115,-13.590,433.291,171.773,27.078,155.026
C03316=1062.121,-13.341,433.278,171.773,27.080,155.026
C03317=1062.127,-13.091,433.264,171.775,27.082,155.026
C03318=1062.134,-12.842,433.250,171.776,27.085,155.027
C03319=1062.139,-12.592,433.236,171.778,27.088,155.027
C03320=1062.146,-12.342,433.222,171.779,27.090,155.027
C03321=1062.152,-12.093,433.208,171.781,27.092,155.028
C03322=1062.158,-11.844,433.194,171.783,27.094,155.028
C03323=1062.164,-11.594,433.180,171.784,27.097,155.028
C03324=1062.170,-11.344,433.166,171.786,27.099,155.028
C03325=1062.176,-11.094,433.152,171.787,27.101,155.029
C03326=1062.182,-10.845,433.138,171.789,27.104,155.029
C03327=1062.188,-10.596,433.124,171.790,27.106,155.029
C03328=1062.194,-10.346,433.110,171.792,27.109,155.030
C03329=1062.201,-10.097,433.096,171.793,27.111,155.030
C03330=1062.206,-9.847,433.082,171.795,27.113,155.030
C03331=1062.212,-9.597,433.068,171.797,27.116,155.030
C03332=1062.219,-9.348,433.054,171.798,27.118,155.031
C03333=1062.225,-9.098,433.040,171.800,27.120,155.031
C03334=1062.230,-8.849,433.025,171.800,27.122,155.031
C03335=1062.237,-8.599,433.012,171.802,27.125,155.032
C03336=1062.243,-8.350,432.998,171.803,27.127,155.032
C03337=1062.249,-8.101,432.983,171.805,27.130,155.032
C03338=1062.255,-7.851,432.970,171.807,27.132,155.032
C03339=1062.261,-7.602,432.955,171.808,27.134,155.033
C03340=1062.267,-7.351,432.941,171.810,27.136,155.033
C03341=1062.273,-7.102,432.927,171.811,27.139,155.033
C03342=1062.280,-6.853,432.912,171.813,27.141,155.034
C03343=1062.285,-6.603,432.899,171.814,27.144,155.034
C03344=1062.292,-6.354,432.884,171.816,27.146,155.034
C03345=1062.298,-6.104,432.870,171.818,27.148,155.034
C03346=1062.304,-5.855,432.856,171.819,27.151,155.035
C03347=1062.310,-5.605,432.842,171.821,27.153,155.035
C03348=1062.316,-5.356,432.828,171.822,27.155,155.035
C03349=1062.322,-5.106,432.813,171.824,27.158,155.036
C03350=1062.328,-4.857,432.799,171.824,27.160,155.036
C03351=1062.335,-4.607,432.785,171.826,27.162,155.036
C03352=1062.341,-4.358,432.771,171.828,27.165,155.036
C03353=1062.347,-4.108,432.756,171.829,27.167,155.037
C03354=1062.353,-3.859,432.742,171.831,27.169,155.037
C03355=1062.359,-3.609,432.728,171.832,27.171,155.037
C03356=1062.366,-3.359,432.713,171.834,27.174,155.038
C03357=1062.371,-3.110,432.699,171.835,27.177,155.038
C03358=1062.377,-2.861,432.685,171.837,27.179,155.038
C03359=1062.383,-2.610,432.671,171.838,27.182,155.039
C03360=1062.390,-2.330,432.654,171.840,27.184,155.039
C03361=1062.397,-2.049,432.638,171.841,27.187,155.039
C03362=1062.404,-1.768,432.621,171.843,27.190,155.040
C03363=1062.411,-1.487,432.606,171.844,27.193,155.040
C03364=1062.416,-1.238,432.591,171.846,27.195,155.040
C03365=1062.422,-0.988,432.577,171.848,27.197,155.040
C03366=1062.428,-0.739,432.562,171.849,27.200,155.041
C03367=1062.434,-0.490,432.548,171.851,27.202,155.041
C03368=1062.440,-0.239,432.533,171.852,27.205,155.041
C03369=1062.446,0.010,432.519,171.854,27.207,155.042
C03370=1062.452,0.259,432.504,171.855,27.210,155.042
C03371=1062.458,0.509,432.490,171.857,27.212,155.042
C03372=1062.464,0.729,432.477,171.858,27.214,155.043
C03373=1062.469,0.949,432.463,171.859,27.216,155.043
C03374=1062.474,1.169,432.451,171.861,27.218,155.043
C03375=1062.479,1.390,432.438,171.862,27.221,155.043
C03376=1062.485,1.609,432.425,171.863,27.223,155.044
C03377=1062.489,1.830,432.412,171.864,27.225,155.044
C03378=1062.495,2.050,432.400,171.866,27.227,155.044
C03379=1062.501,2.270,432.387,171.867,27.229,155.045
C03380=1062.507,2.520,432.372,171.868,27.232,155.045
C03381=1062.512,2.769,432.358,171.870,27.234,155.045
C03382=1062.519,3.019,432.343,171.871,27.237,155.046
C03383=1062.525,3.268,432.328,171.873,27.239,155.046
C03384=1062.531,3.517,432.313,171.874,27.242,155.046
C03385=1062.536,3.767,432.299,171.876,27.244,155.046
C03386=1062.543,4.017,432.284,171.877,27.246,155.047
C03387=1062.549,4.266,432.270,171.879,27.249,155.047
C03388=1062.555,4.515,432.255,171.881,27.252,155.047
C03389=1062.561,4.765,432.240,171.881,27.254,155.048
C03390=1062.567,5.014,432.226,171.883,27.256,155.048
C03391=1062.573,5.264,432.211,171.884,27.259,155.048
C03392=1062.580,5.514,432.196,171.886,27.261,155.049
C03393=1062.585,5.763,432.182,171.887,27.264,155.049
C03394=1062.591,6.013,432.166,171.889,27.266,155.049
C03395=1062.597,6.262,432.152,171.890,27.268,155.050
C03396=1062.603,6.512,432.137,171.892,27.271,155.050
C03397=1062.609,6.762,432.122,171.894,27.273,155.050
C03398=1062.615,7.011,432.108,171.895,27.276,155.051
C03399=1062.621,7.260,432.093,171.897,27.279,155.051
C03400=1062.628,7.510,432.078,171.898,27.281,155.051
C03401=1062.634,7.759,432.063,171.899,27.283,155.052
C03402=1062.640,8.008,432.048,171.900,27.286,155.052
C03403=1062.646,8.257,432.034,171.902,27.288,155.052
C03404=1062.652,8.507,432.019,171.903,27.291,155.053
C03405=1062.659,8.757,432.004,171.905,27.293,155.053
C03406=1062.664,9.006,431.989,171.907,27.295,155.053
C03407=1062.670,9.256,431.975,171.908,27.298,155.053
C03408=1062.677,9.506,431.960,171.910,27.300,155.054
C03409=1062.682,9.756,431.945,171.911,27.303,155.054
C03410=1062.688,10.005,431.930,171.913,27.306,155.054
C03411=1062.695,10.254,431.915,171.914,27.308,155.055
C03412=1062.701,10.504,431.900,171.915,27.310,155.055
C03413=1062.707,10.753,431.886,171.916,27.313,155.055
C03414=1062.713,11.002,431.871,171.918,27.315,155.056
C03415=1062.719,11.252,431.856,171.919,27.318,155.056
C03416=1062.725,11.501,431.841,171.921,27.320,155.056
C03417=1062.732,11.751,431.826,171.923,27.322,155.057
C03418=1062.738,12.000,431.811,171.924,27.325,155.057
C03419=1062.744,12.250,431.796,171.926,27.327,155.057
C03420=1062.749,12.499,431.781,171.927,27.330,155.058
C03421=1062.756,12.748,431.765,171.929,27.333,155.058
C03422=1062.763,12.998,431.750,171.929,27.335,155.058
C03423=1062.769,13.248,431.736,171.931,27.337,155.059
C03424=1062.777,13.589,431.715,171.933,27.341,155.059
C03425=1062.785,13.931,431.694,171.936,27.344,155.059
C03426=1062.795,14.272,431.674,171.937,27.347,155.060
C03427=1062.802,14.613,431.654,171.940,27.351,155.060
C03428=1062.808,14.863,431.638,171.941,27.354,155.061
C03429=1062.814,15.113,431.623,171.943,27.356,155.061
C03430=1062.820,15.362,431.609,171.943,27.358,155.061
C03431=1062.826,15.612,431.593,171.945,27.361,155.062
C03432=1062.832,15.861,431.578,171.946,27.364,155.062
C03433=1062.839,16.110,431.562,171.948,27.366,155.062
C03434=1062.844,16.360,431.547,171.949,27.369,155.063
C03435=1062.850,16.609,431.532,171.951,27.371,155.063
C03436=1062.857,16.859,431.517,171.952,27.374,155.063
C03437=1062.862,17.109,431.502,171.954,27.376,155.064
C03438=1062.868,17.358,431.487,171.956,27.379,155.064
C03439=1062.875,17.607,431.472,171.957,27.381,155.064
C03440=1062.881,17.857,431.456,171.958,27.384,155.065
C03441=1062.887,18.107,431.441,171.959,27.386,155.065
C03442=1062.892,18.356,431.426,171.961,27.389,155.065
C03443=1062.899,18.605,431.410,171.962,27.391,155.066
C03444=1062.905,18.855,431.395,171.964,27.394,155.066
C03445=1062.911,19.105,431.380,171.965,27.396,155.066
C03446=1062.917,19.354,431.365,171.967,27.399,155.067
C03447=1062.923,19.603,431.350,171.969,27.401,155.067
C03448=1062.929,19.853,431.334,171.970,27.404,155.067
C03449=1062.935,20.102,431.319,171.971,27.406,155.068
C03450=1062.941,20.352,431.303,171.972,27.409,155.068
C03451=1062.948,20.601,431.288,171.974,27.411,155.068
C03452=1062.953,20.850,431.273,171.975,27.414,155.069
C03453=1062.959,21.099,431.257,171.977,27.416,155.069
C03454=1062.966,21.349,431.242,171.978,27.419,155.069
C03455=1062.971,21.599,431.227,171.980,27.421,155.070
C03456=1062.978,21.848,431.211,171.981,27.424,155.070
C03457=1062.983,22.097,431.196,171.983,27.427,155.070
C03458=1062.989,22.347,431.181,171.984,27.429,155.071
C03459=1062.995,22.596,431.165,171.985,27.432,155.071
C03460=1063.002,22.846,431.150,171.987,27.434,155.071
C03461=1063.007,23.096,431.134,171.988,27.437,155.072
C03462=1063.013,23.344,431.119,171.990,27.439,155.072
C03463=1063.019,23.594,431.103,171.991,27.442,155.072
C03464=1063.026,23.843,431.088,171.993,27.444,155.073
C03465=1063.031,24.093,431.072,171.994,27.447,155.073
C03466=1063.038,24.342,431.056,171.996,27.450,155.073
C03467=1063.044,24.592,431.041,171.997,27.452,155.074
C03468=1063.050,24.842,431.026,171.998,27.455,155.074
C03469=1063.056,25.091,431.010,172.000,27.457,155.074
C03470=1063.062,25.340,430.995,172.001,27.460,155.075
C03471=1063.068,25.590,430.979,172.003,27.462,155.075
C03472=1063.074,25.840,430.963,172.004,27.465,155.075
C03473=1063.080,26.089,430.948,172.006,27.467,155.076
C03474=1063.086,26.339,430.932,172.007,27.470,155.076
C03475=1063.093,26.588,430.916,172.009,27.473,155.077
C03476=1063.098,26.838,430.901,172.009,27.475,155.077
C03477=1063.105,27.087,430.885,172.011,27.478,155.077
C03478=1063.110,27.336,430.870,172.013,27.480,155.078
C03479=1063.117,27.585,430.854,172.014,27.483,155.078
C03480=1063.122,27.835,430.839,172.016,27.485,155.078
C03481=1063.128,28.084,430.823,172.017,27.488,155.079
C03482=1063.135,28.333,430.807,172.019,27.491,155.079
C03483=1063.141,28.583,430.791,172.020,27.493,155.079
C03484=1063.147,28.832,430.776,172.021,27.496,155.080
C03485=1063.153,29.082,430.760,172.022,27.498,155.080
C03486=1063.159,29.332,430.744,172.024,27.501,155.080
C03487=1063.164,29.582,430.728,172.025,27.504,155.081
C03488=1063.172,29.866,430.710,172.027,27.506,155.081
C03489=1063.178,30.149,430.693,172.028,27.509,155.082
C03490=1063.185,30.434,430.675,172.031,27.512,155.082
C03491=1063.192,30.717,430.657,172.032,27.515,155.082
C03492=1063.198,30.967,430.640,172.034,27.518,155.083
C03493=1063.203,31.217,430.625,172.034,27.521,155.083
C03494=1063.210,31.466,430.609,172.036,27.523,155.083
C03495=1063.216,31.715,430.593,172.038,27.526,155.084
C03496=1063.222,31.965,430.577,172.039,27.528,155.084
C03497=1063.228,32.214,430.561,172.041,27.531,155.084
C03498=1063.234,32.463,430.546,172.042,27.534,155.085
C03499=1063.240,32.713,430.530,172.044,27.536,155.085
C03500=1063.246,32.963,430.514,172.045,27.539,155.085
C03501=1063.252,33.212,430.497,172.046,27.541,155.086
C03502=1063.259,33.461,430.482,172.047,27.544,155.086
C03503=1063.264,33.711,430.466,172.049,27.546,155.087
C03504=1063.270,33.960,430.450,172.050,27.549,155.087
C03505=1063.276,34.210,430.434,172.052,27.552,155.087
C03506=1063.283,34.459,430.418,172.054,27.554,155.088
C03507=1063.288,34.709,430.403,172.055,27.557,155.088
C03508=1063.294,34.958,430.386,172.057,27.559,155.088
C03509=1063.300,35.208,430.370,172.057,27.562,155.089
C03510=1063.306,35.457,430.354,172.059,27.565,155.089
C03511=1063.313,35.707,430.339,172.060,27.567,155.089
C03512=1063.319,35.956,430.323,172.062,27.570,155.090
C03513=1063.325,36.205,430.306,172.063,27.573,155.090
C03514=1063.331,36.455,430.290,172.065,27.575,155.090
C03515=1063.337,36.704,430.274,172.067,27.578,155.091
C03516=1063.343,36.953,430.258,172.068,27.580,155.091
C03517=1063.349,37.203,430.243,172.070,27.583,155.092
C03518=1063.355,37.452,430.226,172.070,27.585,155.092
C03519=1063.361,37.702,430.210,172.072,27.588,155.092
C03520=1063.367,37.951,430.194,172.073,27.590,155.093
C03521=1063.373,38.200,430.178,172.075,27.593,155.093
C03522=1063.379,38.449,430.162,172.076,27.596,155.093
C03523=1063.385,38.699,430.146,172.078,27.598,155.094
C03524=1063.391,38.948,430.129,172.079,27.601,155.094
C03525=1063.397,39.198,430.114,172.081,27.604,155.094
C03526=1063.403,39.447,430.098,172.082,27.606,155.095
C03527=1063.409,39.697,430.081,172.083,27.609,155.095
C03528=1063.415,39.946,430.065,172.085,27.612,155.096
C03529=1063.421,40.195,430.049,172.086,27.614,155.096
C03530=1063.427,40.445,430.033,172.088,27.617,155.096
C03531=1063.433,40.694,430.016,172.089,27.619,155.097
C03532=1063.439,40.943,430.000,172.091,27.622,155.097
C03533=1063.444,41.193,429.984,172.092,27.625,155.097
C03534=1063.450,41.442,429.968,172.093,27.627,155.098
C03535=1063.456,41.691,429.951,172.095,27.630,155.098
C03536=1063.462,41.941,429.935,172.096,27.633,155.098
C03537=1063.469,42.191,429.918,172.098,27.636,155.099
C03538=1063.475,42.440,429.902,172.099,27.638,155.099
C03539=1063.481,42.690,429.886,172.101,27.641,155.100
C03540=1063.487,42.939,429.870,172.102,27.643,155.100
C03541=1063.493,43.188,429.853,172.104,27.646,155.100
C03542=1063.499,43.438,429.837,172.104,27.648,155.101
C03543=1063.505,43.687,429.821,172.106,27.651,155.101
C03544=1063.510,43.937,429.804,172.107,27.654,155.101
C03545=1063.516,44.186,429.788,172.109,27.657,155.102
C03546=1063.522,44.435,429.772,172.111,27.659,155.102
C03547=1063.528,44.684,429.755,172.112,27.662,155.103
C03548=1063.534,44.933,429.738,172.114,27.665,155.103
C03549=1063.539,45.183,429.721,172.114,27.667,155.103
C03550=1063.545,45.432,429.705,172.116,27.670,155.104
C03551=1063.552,45.682,429.689,172.117,27.673,155.104
C03552=1063.558,45.967,429.670,172.119,27.676,155.105
C03553=1063.565,46.251,429.651,172.120,27.678,155.105
C03554=1063.571,46.534,429.632,172.123,27.682,155.105
C03555=1063.578,46.819,429.613,172.124,27.685,155.106
C03556=1063.584,47.068,429.597,172.126,27.688,155.106
C03557=1063.590,47.317,429.581,172.126,27.690,155.107
C03558=1063.595,47.566,429.563,172.128,27.693,155.107
C03559=1063.602,47.816,429.547,172.129,27.695,155.107
C03560=1063.608,48.066,429.530,172.131,27.698,155.108
C03561=1063.614,48.315,429.514,172.132,27.701,155.108
C03562=1063.619,48.565,429.497,172.134,27.704,155.108
C03563=1063.625,48.813,429.480,172.135,27.707,155.109
C03564=1063.631,49.063,429.464,172.137,27.709,155.109
C03565=1063.637,49.312,429.448,172.138,27.711,155.110
C03566=1063.642,49.562,429.431,172.139,27.714,155.110
C03567=1063.649,49.811,429.414,172.141,27.717,155.110
C03568=1063.655,50.061,429.397,172.142,27.720,155.111
C03569=1063.660,50.310,429.381,172.144,27.722,155.111
C03570=1063.666,50.560,429.364,172.145,27.725,155.111
C03571=1063.673,50.808,429.347,172.147,27.728,155.112
C03572=1063.679,51.058,429.331,172.148,27.731,155.112
C03573=1063.684,51.308,429.314,172.149,27.733,155.113
C03574=1063.691,51.557,429.297,172.150,27.736,155.113
C03575=1063.697,51.806,429.281,172.152,27.738,155.113
C03576=1063.703,52.056,429.264,172.154,27.741,155.114
C03577=1063.708,52.305,429.247,172.155,27.744,155.114
C03578=1063.715,52.555,429.230,172.157,27.747,155.114
C03579=1063.721,52.804,429.214,172.158,27.749,155.115
C03580=1063.726,53.053,429.196,172.160,27.752,155.115
C03581=1063.732,53.302,429.180,172.160,27.754,155.116
C03582=1063.738,53.552,429.164,172.162,27.757,155.116
C03583=1063.744,53.801,429.146,172.163,27.760,155.116
C03584=1063.750,54.051,429.130,172.165,27.762,155.117
C03585=1063.756,54.299,429.113,172.167,27.765,155.117
C03586=1063.762,54.549,429.096,172.168,27.768,155.117
C03587=1063.768,54.799,429.079,172.170,27.770,155.118
C03588=1063.774,55.048,429.062,172.171,27.773,155.118
C03589=1063.780,55.297,429.046,172.172,27.775,155.119
C03590=1063.786,55.546,429.028,172.173,27.778,155.119
C03591=1063.792,55.796,429.012,172.175,27.781,155.119
C03592=1063.799,56.045,428.995,172.176,27.784,155.120
C03593=1063.804,56.295,428.978,172.178,27.786,155.120
C03594=1063.810,56.544,428.962,172.180,27.789,155.120
C03595=1063.817,56.794,428.944,172.181,27.792,155.121
C03596=1063.822,57.043,428.927,172.183,27.794,155.121
C03597=1063.828,57.292,428.911,172.183,27.797,155.122
C03598=1063.835,57.542,428.894,172.185,27.799,155.122
C03599=1063.840,57.791,428.876,172.186,27.802,155.122
C03600=1063.846,58.040,428.860,172.188,27.805,155.123
C03601=1063.852,58.289,428.843,172.189,27.808,155.123
C03602=1063.859,58.539,428.825,172.191,27.810,155.123
C03603=1063.864,58.788,428.809,172.193,27.813,155.124
C03604=1063.870,59.037,428.791,172.194,27.815,155.124
C03605=1063.877,59.287,428.775,172.195,27.818,155.125
C03606=1063.883,59.536,428.758,172.196,27.820,155.125
C03607=1063.888,59.786,428.741,172.198,27.823,155.125
C03608=1063.895,60.035,428.724,172.199,27.826,155.126
C03609=1063.901,60.284,428.707,172.201,27.829,155.126
C03610=1063.906,60.533,428.690,172.203,27.831,155.126
C03611=1063.913,60.783,428.672,172.204,27.834,155.127
C03612=1063.919,61.032,428.656,172.206,27.836,155.127
C03613=1063.925,61.282,428.638,172.207,27.839,155.128
C03614=1063.931,61.531,428.622,172.208,27.841,155.128
C03615=1063.937,61.780,428.604,172.209,27.844,155.128
C03616=1063.944,62.065,428.585,172.211,27.847,155.129
C03617=1063.951,62.348,428.565,172.213,27.850,155.129
C03618=1063.958,62.632,428.546,172.215,27.853,155.129
C03619=1063.965,62.916,428.526,172.216,27.856,155.130
C03620=1063.971,63.165,428.509,172.218,27.859,155.130
C03621=1063.977,63.415,428.492,172.220,27.861,155.131
C03622=1063.984,63.664,428.475,172.221,27.864,155.131
C03623=1063.989,63.913,428.458,172.222,27.866,155.131
C03624=1063.996,64.163,428.441,172.223,27.869,155.132
C03625=1064.002,64.412,428.424,172.225,27.872,155.132
C03626=1064.008,64.661,428.406,172.226,27.874,155.132
C03627=1064.013,64.911,428.389,172.228,27.877,155.133
C03628=1064.019,65.160,428.372,172.229,27.880,155.133
C03629=1064.026,65.410,428.354,172.231,27.883,155.134
C03630=1064.031,65.659,428.337,172.233,27.886,155.134
C03631=1064.037,65.907,428.320,172.234,27.888,155.134
C03632=1064.043,66.158,428.303,172.235,27.890,155.135
C03633=1064.049,66.406,428.286,172.236,27.893,155.135
C03634=1064.056,66.656,428.268,172.238,27.896,155.136
C03635=1064.061,66.905,428.250,172.239,27.899,155.136
C03636=1064.067,67.154,428.233,172.241,27.902,155.136
C03637=1064.073,67.404,428.216,172.243,27.904,155.137
